gfCNCPoint3[13260] = {X 553.8289, Y 64.3705, Z -4.6667, A 0.000, B 0.000, C 0.000 }
gfCNCPoint3[13261] = {X 551.8531, Y 63.3648, Z -4.6667, A 0.000, B 0.000, C 0.000 }
gfCNCPoint3[13262] = {X 549.9931, Y 62.1583, Z -4.6667, A 0.000, B 0.000, C 0.000 }
gfCNCPoint3[13263] = {X 548.2693, Y 60.7642, Z -4.6667, A 0.000, B 0.000, C 0.000 }
gfCNCPoint3[13264] = {X 546.7005, Y 59.1977, Z -4.6667, A 0.000, B 0.000, C 0.000 }
gfCNCPoint3[13265] = {X 545.1840, Y 59.4175, Z -4.6667, A 0.000, B 0.000, C 0.000 }
gfCNCPoint3[13266] = {X 543.6528, Y 59.4759, Z -4.6667, A 0.000, B 0.000, C 0.000 }
gfCNCPoint3[13267] = {X 527.5783, Y 59.4763, Z -4.6667, A 0.000, B 0.000, C 0.000 }
gfCNCPoint3[13268] = {X 525.9215, Y 60.2766, Z -4.6667, A 0.000, B 0.000, C 0.000 }
gfCNCPoint3[13269] = {X 524.1774, Y 60.8627, Z -4.6667, A 0.000, B 0.000, C 0.000 }
gfCNCPoint3[13270] = {X 522.3736, Y 61.2254, Z -4.6667, A 0.000, B 0.000, C 0.000 }
gfCNCPoint3[13271] = {X 520.5385, Y 61.3590, Z -4.6667, A 0.000, B 0.000, C 0.000 }
gfCNCPoint3[13272] = {X 519.7998, Y 61.3591, Z -4.6667, A 0.000, B 0.000, C 0.000 }
gfCNCPoint3[13273] = {X 518.0043, Y 61.2474, Z -4.6667, A 0.000, B 0.000, C 0.000 }
gfCNCPoint3[13274] = {X 516.2365, Y 60.9138, Z -4.6667, A 0.000, B 0.000, C 0.000 }
gfCNCPoint3[13275] = {X 514.5237, Y 60.3637, Z -4.6667, A 0.000, B 0.000, C 0.000 }
gfCNCPoint3[13276] = {X 512.8923, Y 59.6054, Z -4.6667, A 0.000, B 0.000, C 0.000 }
gfCNCPoint3[13277] = {X 511.3676, Y 58.6507, Z -4.6667, A 0.000, B 0.000, C 0.000 }
gfCNCPoint3[13278] = {X 509.9730, Y 57.5142, Z -4.6667, A 0.000, B 0.000, C 0.000 }
gfCNCPoint3[13279] = {X 508.6156, Y 58.2113, Z -4.6667, A 0.000, B 0.000, C 0.000 }
gfCNCPoint3[13280] = {X 507.1924, Y 58.7617, Z -4.6667, A 0.000, B 0.000, C 0.000 }
gfCNCPoint3[13281] = {X 505.7192, Y 59.1593, Z -4.6667, A 0.000, B 0.000, C 0.000 }
gfCNCPoint3[13282] = {X 504.2123, Y 59.3996, Z -4.6667, A 0.000, B 0.000, C 0.000 }
gfCNCPoint3[13283] = {X 502.6885, Y 59.4800, Z -4.6667, A 0.000, B 0.000, C 0.000 }
gfCNCPoint3[13284] = {X 496.2450, Y 59.4800, Z -4.6667, A 0.000, B 0.000, C 0.000 }
gfCNCPoint3[13285] = {X 495.2580, Y 59.4463, Z -4.6667, A 0.000, B 0.000, C 0.000 }
gfCNCPoint3[13286] = {X 494.2756, Y 59.3454, Z -4.6667, A 0.000, B 0.000, C 0.000 }
gfCNCPoint3[13287] = {X 494.1342, Y 61.3005, Z -4.6667, A 0.000, B 0.000, C 0.000 }
gfCNCPoint3[13288] = {X 493.7950, Y 63.2312, Z -4.6667, A 0.000, B 0.000, C 0.000 }
gfCNCPoint3[13289] = {X 493.2616, Y 65.1174, Z -4.6667, A 0.000, B 0.000, C 0.000 }
gfCNCPoint3[13290] = {X 492.5393, Y 66.9397, Z -4.6667, A 0.000, B 0.000, C 0.000 }
gfCNCPoint3[13291] = {X 491.6358, Y 68.6792, Z -4.6667, A 0.000, B 0.000, C 0.000 }
gfCNCPoint3[13292] = {X 490.5603, Y 70.3180, Z -4.6667, A 0.000, B 0.000, C 0.000 }
gfCNCPoint3[13293] = {X 490.5605, Y 83.2950, Z -4.6667, A 0.000, B 0.000, C 0.000 }
gfCNCPoint3[13294] = {X 507.6815, Y 83.2950, Z -4.6667, A 0.000, B 0.000, C 0.000 }
gfCNCPoint3[13295] = {X 507.6815, Y 85.6950, Z -4.6667, A 0.000, B 0.000, C 0.000 }
gfCNCPoint3[13296] = {X 585.6966, Y 85.6950, Z -4.6667, A 0.000, B 0.000, C 0.000 }
gfCNCPoint3[13297] = {X 585.6966, Y 63.3150, Z -4.6667, A 0.000, B 0.000, C 0.000 }
gfCNCPoint3[13298] = {X 584.3995, Y 63.5678, Z -4.6667, A 0.000, B 0.000, C 0.000 }
gfCNCPoint3[13299] = {X 583.0880, Y 63.7288, Z -4.6667, A 0.000, B 0.000, C 0.000 }
gfCNCPoint3[13300] = {X 581.1243, Y 63.7971, Z -4.6667, A 0.000, B 0.000, C 0.000 }
gfCNCPoint3[13301] = {X 579.1642, Y 63.6600, Z -4.6667, A 0.000, B 0.000, C 0.000 }
gfCNCPoint3[13302] = {X 577.2291, Y 63.3191, Z -4.6667, A 0.000, B 0.000, C 0.000 }
gfCNCPoint3[13303] = {X 575.3401, Y 62.7781, Z -4.6667, A 0.000, B 0.000, C 0.000 }
gfCNCPoint3[13304] = {X 573.3441, Y 63.3435, Z -4.6667, A 0.000, B 0.000, C 0.000 }
gfCNCPoint3[13305] = {X 571.2979, Y 63.6855, Z -4.6667, A 0.000, B 0.000, C 0.000 }
gfCNCPoint3[13306] = {X 569.2264, Y 63.8000, Z -4.6667, A 0.000, B 0.000, C 0.000 }
gfCNCPoint3[13307] = {X 562.4443, Y 63.8000, Z -4.6667, A 0.000, B 0.000, C 0.000 }
gfCNCPoint3[13308] = {X 560.5408, Y 63.7034, Z -4.6667, A 0.000, B 0.000, C 0.000 }
gfCNCPoint3[13309] = {X 558.6568, Y 63.4145, Z -4.6667, A 0.000, B 0.000, C 0.000 }
gfCNCPoint3[13310] = {X 556.8118, Y 62.9364, Z -4.6667, A 0.000, B 0.000, C 0.000 }
gfCNCPoint3[13311] = {X 555.0247, Y 62.2739, Z -4.6667, A 0.000, B 0.000, C 0.000 }
gfCNCPoint3[13312] = {X 553.3138, Y 61.4339, Z -4.6667, A 0.000, B 0.000, C 0.000 }
gfCNCPoint3[13313] = {X 551.6968, Y 60.4250, Z -4.6667, A 0.000, B 0.000, C 0.000 }
gfCNCPoint3[13314] = {X 550.1902, Y 59.2575, Z -4.6667, A 0.000, B 0.000, C 0.000 }
gfCNCPoint3[13315] = {X 548.8096, Y 57.9435, Z -4.6667, A 0.000, B 0.000, C 0.000 }
gfCNCPoint3[13316] = {X 547.5691, Y 56.4965, Z -4.6667, A 0.000, B 0.000, C 0.000 }
gfCNCPoint3[13317] = {X 546.2936, Y 56.8314, Z -4.6667, A 0.000, B 0.000, C 0.000 }
gfCNCPoint3[13318] = {X 544.9891, Y 57.0253, Z -4.6667, A 0.000, B 0.000, C 0.000 }
gfCNCPoint3[13319] = {X 543.6713, Y 57.0759, Z -4.6667, A 0.000, B 0.000, C 0.000 }
gfCNCPoint3[13320] = {X 526.9187, Y 57.0763, Z -4.6667, A 0.000, B 0.000, C 0.000 }
gfCNCPoint3[13321] = {X 525.4335, Y 57.8746, Z -4.6667, A 0.000, B 0.000, C 0.000 }
gfCNCPoint3[13322] = {X 523.8527, Y 58.4612, Z -4.6667, A 0.000, B 0.000, C 0.000 }
gfCNCPoint3[13323] = {X 522.2063, Y 58.8250, Z -4.6667, A 0.000, B 0.000, C 0.000 }
gfCNCPoint3[13324] = {X 520.5255, Y 58.9590, Z -4.6667, A 0.000, B 0.000, C 0.000 }
gfCNCPoint3[13325] = {X 519.7998, Y 58.9591, Z -4.6667, A 0.000, B 0.000, C 0.000 }
gfCNCPoint3[13326] = {X 518.2467, Y 58.8589, Z -4.6667, A 0.000, B 0.000, C 0.000 }
gfCNCPoint3[13327] = {X 516.7195, Y 58.5598, Z -4.6667, A 0.000, B 0.000, C 0.000 }
gfCNCPoint3[13328] = {X 515.2433, Y 58.0668, Z -4.6667, A 0.000, B 0.000, C 0.000 }
gfCNCPoint3[13329] = {X 513.8428, Y 57.3882, Z -4.6667, A 0.000, B 0.000, C 0.000 }
gfCNCPoint3[13330] = {X 512.5411, Y 56.5351, Z -4.6667, A 0.000, B 0.000, C 0.000 }
gfCNCPoint3[13331] = {X 511.3600, Y 55.5218, Z -4.6667, A 0.000, B 0.000, C 0.000 }
gfCNCPoint3[13332] = {X 510.3189, Y 54.3650, Z -4.6667, A 0.000, B 0.000, C 0.000 }
gfCNCPoint3[13333] = {X 508.9711, Y 55.3177, Z -4.6667, A 0.000, B 0.000, C 0.000 }
gfCNCPoint3[13334] = {X 507.5060, Y 56.0778, Z -4.6667, A 0.000, B 0.000, C 0.000 }
gfCNCPoint3[13335] = {X 505.9510, Y 56.6311, Z -4.6667, A 0.000, B 0.000, C 0.000 }
gfCNCPoint3[13336] = {X 504.3351, Y 56.9672, Z -4.6667, A 0.000, B 0.000, C 0.000 }
gfCNCPoint3[13337] = {X 502.6885, Y 57.0800, Z -4.6667, A 0.000, B 0.000, C 0.000 }
gfCNCPoint3[13338] = {X 496.2450, Y 57.0800, Z -4.6667, A 0.000, B 0.000, C 0.000 }
gfCNCPoint3[13339] = {X 495.4216, Y 57.0519, Z -4.6667, A 0.000, B 0.000, C 0.000 }
gfCNCPoint3[13340] = {X 494.6020, Y 56.9677, Z -4.6667, A 0.000, B 0.000, C 0.000 }
gfCNCPoint3[13341] = {X 493.1719, Y 56.6826, Z -4.6667, A 0.000, B 0.000, C 0.000 }
gfCNCPoint3[13342] = {X 491.7866, Y 56.2272, Z -4.6667, A 0.000, B 0.000, C 0.000 }
gfCNCPoint3[13343] = {X 491.8566, Y 57.1124, Z -4.6667, A 0.000, B 0.000, C 0.000 }
gfCNCPoint3[13344] = {X 491.8800, Y 58.0000, Z -4.6667, A 0.000, B 0.000, C 0.000 }
gfCNCPoint3[13345] = {X 491.8794, Y 59.0735, Z -4.6667, A 0.000, B 0.000, C 0.000 }
gfCNCPoint3[13346] = {X 491.8781, Y 59.1839, Z -4.6667, A 0.000, B 0.000, C 0.000 }
gfCNCPoint3[13347] = {X 491.8762, Y 59.2942, Z -4.6667, A 0.000, B 0.000, C 0.000 }
gfCNCPoint3[13348] = {X 491.7363, Y 61.1318, Z -4.6667, A 0.000, B 0.000, C 0.000 }
gfCNCPoint3[13349] = {X 491.3970, Y 62.9431, Z -4.6667, A 0.000, B 0.000, C 0.000 }
gfCNCPoint3[13350] = {X 490.8623, Y 64.7067, Z -4.6667, A 0.000, B 0.000, C 0.000 }
gfCNCPoint3[13351] = {X 490.1385, Y 66.4014, Z -4.6667, A 0.000, B 0.000, C 0.000 }
gfCNCPoint3[13352] = {X 489.2342, Y 68.0072, Z -4.6667, A 0.000, B 0.000, C 0.000 }
gfCNCPoint3[13353] = {X 488.1603, Y 69.5048, Z -4.6667, A 0.000, B 0.000, C 0.000 }
gfCNCPoint3[13354] = {X 488.1606, Y 85.6950, Z -4.6667, A 0.000, B 0.000, C 0.000 }
gfCNCPoint3[13355] = {X 507.6815, Y 85.6950, Z -4.6667, A 0.000, B 0.000, C 0.000 }
gfCNCPoint3[13356] = {X 507.6815, Y 88.0950, Z -4.6667, A 0.000, B 0.000, C 0.000 }
gfCNCPoint3[13357] = {X 588.0966, Y 88.0950, Z -4.6667, A 0.000, B 0.000, C 0.000 }
gfCNCPoint3[13358] = {X 588.0966, Y 60.4644, Z -4.6667, A 0.000, B 0.000, C 0.000 }
gfCNCPoint3[13359] = {X 587.7998, Y 60.3564, Z -4.6667, A 0.000, B 0.000, C 0.000 }
gfCNCPoint3[13360] = {X 587.5052, Y 60.2427, Z -4.6667, A 0.000, B 0.000, C 0.000 }
gfCNCPoint3[13361] = {X 586.3439, Y 60.6540, Z -4.6667, A 0.000, B 0.000, C 0.000 }
gfCNCPoint3[13362] = {X 585.1550, Y 60.9769, Z -4.6667, A 0.000, B 0.000, C 0.000 }
gfCNCPoint3[13363] = {X 583.5153, Y 61.2699, Z -4.6667, A 0.000, B 0.000, C 0.000 }
gfCNCPoint3[13364] = {X 581.8543, Y 61.3951, Z -4.6667, A 0.000, B 0.000, C 0.000 }
gfCNCPoint3[13365] = {X 580.1893, Y 61.3512, Z -4.6667, A 0.000, B 0.000, C 0.000 }
gfCNCPoint3[13366] = {X 578.5372, Y 61.1386, Z -4.6667, A 0.000, B 0.000, C 0.000 }
gfCNCPoint3[13367] = {X 576.9153, Y 60.7595, Z -4.6667, A 0.000, B 0.000, C 0.000 }
gfCNCPoint3[13368] = {X 575.3401, Y 60.2178, Z -4.6667, A 0.000, B 0.000, C 0.000 }
gfCNCPoint3[13369] = {X 573.8611, Y 60.7315, Z -4.6667, A 0.000, B 0.000, C 0.000 }
gfCNCPoint3[13370] = {X 572.3399, Y 61.1017, Z -4.6667, A 0.000, B 0.000, C 0.000 }
gfCNCPoint3[13371] = {X 570.7903, Y 61.3253, Z -4.6667, A 0.000, B 0.000, C 0.000 }
gfCNCPoint3[13372] = {X 569.2264, Y 61.4000, Z -4.6667, A 0.000, B 0.000, C 0.000 }
gfCNCPoint3[13373] = {X 562.4443, Y 61.4000, Z -4.6667, A 0.000, B 0.000, C 0.000 }
gfCNCPoint3[13374] = {X 560.5829, Y 61.2940, Z -4.6667, A 0.000, B 0.000, C 0.000 }
gfCNCPoint3[13375] = {X 558.7455, Y 60.9774, Z -4.6667, A 0.000, B 0.000, C 0.000 }
gfCNCPoint3[13376] = {X 556.9559, Y 60.4544, Z -4.6667, A 0.000, B 0.000, C 0.000 }
gfCNCPoint3[13377] = {X 555.2372, Y 59.7315, Z -4.6667, A 0.000, B 0.000, C 0.000 }
gfCNCPoint3[13378] = {X 553.6118, Y 58.8183, Z -4.6667, A 0.000, B 0.000, C 0.000 }
gfCNCPoint3[13379] = {X 552.1004, Y 57.7265, Z -4.6667, A 0.000, B 0.000, C 0.000 }
gfCNCPoint3[13380] = {X 550.7228, Y 56.4702, Z -4.6667, A 0.000, B 0.000, C 0.000 }
gfCNCPoint3[13381] = {X 549.4966, Y 55.0657, Z -4.6667, A 0.000, B 0.000, C 0.000 }
gfCNCPoint3[13382] = {X 548.4378, Y 53.5310, Z -4.6667, A 0.000, B 0.000, C 0.000 }
gfCNCPoint3[13383] = {X 547.3159, Y 54.0426, Z -4.6667, A 0.000, B 0.000, C 0.000 }
gfCNCPoint3[13384] = {X 546.1381, Y 54.4074, Z -4.6667, A 0.000, B 0.000, C 0.000 }
gfCNCPoint3[13385] = {X 544.9235, Y 54.6197, Z -4.6667, A 0.000, B 0.000, C 0.000 }
gfCNCPoint3[13386] = {X 543.6918, Y 54.6759, Z -4.6667, A 0.000, B 0.000, C 0.000 }
gfCNCPoint3[13387] = {X 526.1843, Y 54.6763, Z -4.6667, A 0.000, B 0.000, C 0.000 }
gfCNCPoint3[13388] = {X 524.8902, Y 55.4730, Z -4.6667, A 0.000, B 0.000, C 0.000 }
gfCNCPoint3[13389] = {X 523.4888, Y 56.0608, Z -4.6667, A 0.000, B 0.000, C 0.000 }
gfCNCPoint3[13390] = {X 522.0136, Y 56.4257, Z -4.6667, A 0.000, B 0.000, C 0.000 }
gfCNCPoint3[13391] = {X 520.4998, Y 56.5591, Z -4.6667, A 0.000, B 0.000, C 0.000 }
gfCNCPoint3[13392] = {X 519.7998, Y 56.5591, Z -4.6667, A 0.000, B 0.000, C 0.000 }
gfCNCPoint3[13393] = {X 518.3493, Y 56.4498, Z -4.6667, A 0.000, B 0.000, C 0.000 }
gfCNCPoint3[13394] = {X 516.9316, Y 56.1244, Z -4.6667, A 0.000, B 0.000, C 0.000 }
gfCNCPoint3[13395] = {X 515.5787, Y 55.5903, Z -4.6667, A 0.000, B 0.000, C 0.000 }
gfCNCPoint3[13396] = {X 514.3210, Y 54.8595, Z -4.6667, A 0.000, B 0.000, C 0.000 }
gfCNCPoint3[13397] = {X 513.1871, Y 53.9484, Z -4.6667, A 0.000, B 0.000, C 0.000 }
gfCNCPoint3[13398] = {X 512.2025, Y 52.8778, Z -4.6667, A 0.000, B 0.000, C 0.000 }
gfCNCPoint3[13399] = {X 511.3855, Y 51.6648, Z -4.6667, A 0.000, B 0.000, C 0.000 }
gfCNCPoint3[13400] = {X 510.7606, Y 50.3426, Z -4.6667, A 0.000, B 0.000, C 0.000 }
gfCNCPoint3[13401] = {X 509.8636, Y 51.4977, Z -4.6667, A 0.000, B 0.000, C 0.000 }
gfCNCPoint3[13402] = {X 508.8029, Y 52.5044, Z -4.6667, A 0.000, B 0.000, C 0.000 }
gfCNCPoint3[13403] = {X 507.7229, Y 53.2678, Z -4.6667, A 0.000, B 0.000, C 0.000 }
gfCNCPoint3[13404] = {X 506.5489, Y 53.8769, Z -4.6667, A 0.000, B 0.000, C 0.000 }
gfCNCPoint3[13405] = {X 505.3028, Y 54.3203, Z -4.6667, A 0.000, B 0.000, C 0.000 }
gfCNCPoint3[13406] = {X 504.0080, Y 54.5896, Z -4.6667, A 0.000, B 0.000, C 0.000 }
gfCNCPoint3[13407] = {X 502.6885, Y 54.6800, Z -4.6667, A 0.000, B 0.000, C 0.000 }
gfCNCPoint3[13408] = {X 496.2450, Y 54.6800, Z -4.6667, A 0.000, B 0.000, C 0.000 }
gfCNCPoint3[13409] = {X 495.0285, Y 54.6033, Z -4.6667, A 0.000, B 0.000, C 0.000 }
gfCNCPoint3[13410] = {X 493.8313, Y 54.3742, Z -4.6667, A 0.000, B 0.000, C 0.000 }
gfCNCPoint3[13411] = {X 492.6724, Y 53.9966, Z -4.6667, A 0.000, B 0.000, C 0.000 }
gfCNCPoint3[13412] = {X 491.4451, Y 53.4062, Z -4.6667, A 0.000, B 0.000, C 0.000 }
gfCNCPoint3[13413] = {X 490.3129, Y 52.6493, Z -4.6667, A 0.000, B 0.000, C 0.000 }
gfCNCPoint3[13414] = {X 489.2980, Y 51.7410, Z -4.6667, A 0.000, B 0.000, C 0.000 }
gfCNCPoint3[13415] = {X 488.8683, Y 52.1573, Z -4.6667, A 0.000, B 0.000, C 0.000 }
gfCNCPoint3[13416] = {X 488.4137, Y 52.5463, Z -4.6667, A 0.000, B 0.000, C 0.000 }
gfCNCPoint3[13417] = {X 488.8649, Y 53.8245, Z -4.6667, A 0.000, B 0.000, C 0.000 }
gfCNCPoint3[13418] = {X 489.1946, Y 55.1393, Z -4.6667, A 0.000, B 0.000, C 0.000 }
gfCNCPoint3[13419] = {X 489.3999, Y 56.4792, Z -4.6667, A 0.000, B 0.000, C 0.000 }
gfCNCPoint3[13420] = {X 489.4600, Y 57.2386, Z -4.6667, A 0.000, B 0.000, C 0.000 }
gfCNCPoint3[13421] = {X 489.4800, Y 58.0000, Z -4.6667, A 0.000, B 0.000, C 0.000 }
gfCNCPoint3[13422] = {X 489.4795, Y 59.0537, Z -4.6667, A 0.000, B 0.000, C 0.000 }
gfCNCPoint3[13423] = {X 489.3596, Y 60.7977, Z -4.6667, A 0.000, B 0.000, C 0.000 }
gfCNCPoint3[13424] = {X 489.0303, Y 62.5146, Z -4.6667, A 0.000, B 0.000, C 0.000 }
gfCNCPoint3[13425] = {X 488.4966, Y 64.1793, Z -4.6667, A 0.000, B 0.000, C 0.000 }
gfCNCPoint3[13426] = {X 487.7661, Y 65.7676, Z -4.6667, A 0.000, B 0.000, C 0.000 }
gfCNCPoint3[13427] = {X 486.8496, Y 67.2562, Z -4.6667, A 0.000, B 0.000, C 0.000 }
gfCNCPoint3[13428] = {X 485.7603, Y 68.6236, Z -4.6667, A 0.000, B 0.000, C 0.000 }
gfCNCPoint3[13429] = {X 485.7606, Y 87.3794, Z -4.6667, A 0.000, B 0.000, C 0.000 }
gfCNCPoint3[13430] = {X 486.0686, Y 87.7323, Z -4.6667, A 0.000, B 0.000, C 0.000 }
gfCNCPoint3[13431] = {X 486.3650, Y 88.0950, Z -4.6667, A 0.000, B 0.000, C 0.000 }
gfCNCPoint3[13432] = {X 507.6815, Y 88.0950, Z -4.6667, A 0.000, B 0.000, C 0.000 }
gfCNCPoint3[13433] = {X 507.6815, Y 90.4950, Z -4.6667, A 0.000, B 0.000, C 0.000 }
gfCNCPoint3[13434] = {X 590.4966, Y 90.4950, Z -4.6667, A 0.000, B 0.000, C 0.000 }
gfCNCPoint3[13435] = {X 590.4966, Y 58.6615, Z -4.6667, A 0.000, B 0.000, C 0.000 }
gfCNCPoint3[13436] = {X 588.9715, Y 58.2279, Z -4.6667, A 0.000, B 0.000, C 0.000 }
gfCNCPoint3[13437] = {X 587.5052, Y 57.6246, Z -4.6667, A 0.000, B 0.000, C 0.000 }
gfCNCPoint3[13438] = {X 585.8387, Y 58.2956, Z -4.6667, A 0.000, B 0.000, C 0.000 }
gfCNCPoint3[13439] = {X 584.0999, Y 58.7477, Z -4.6667, A 0.000, B 0.000, C 0.000 }
gfCNCPoint3[13440] = {X 582.3176, Y 58.9733, Z -4.6667, A 0.000, B 0.000, C 0.000 }
gfCNCPoint3[13441] = {X 580.5210, Y 58.9689, Z -4.6667, A 0.000, B 0.000, C 0.000 }
gfCNCPoint3[13442] = {X 578.7398, Y 58.7344, Z -4.6667, A 0.000, B 0.000, C 0.000 }
gfCNCPoint3[13443] = {X 577.0034, Y 58.2738, Z -4.6667, A 0.000, B 0.000, C 0.000 }
gfCNCPoint3[13444] = {X 575.3401, Y 57.5945, Z -4.6667, A 0.000, B 0.000, C 0.000 }
gfCNCPoint3[13445] = {X 573.8813, Y 58.2035, Z -4.6667, A 0.000, B 0.000, C 0.000 }
gfCNCPoint3[13446] = {X 572.3630, Y 58.6441, Z -4.6667, A 0.000, B 0.000, C 0.000 }
gfCNCPoint3[13447] = {X 570.8048, Y 58.9107, Z -4.6667, A 0.000, B 0.000, C 0.000 }
gfCNCPoint3[13448] = {X 569.2264, Y 59.0000, Z -4.6667, A 0.000, B 0.000, C 0.000 }
gfCNCPoint3[13449] = {X 562.4443, Y 59.0000, Z -4.6667, A 0.000, B 0.000, C 0.000 }
gfCNCPoint3[13450] = {X 560.6577, Y 58.8855, Z -4.6667, A 0.000, B 0.000, C 0.000 }
gfCNCPoint3[13451] = {X 558.9002, Y 58.5440, Z -4.6667, A 0.000, B 0.000, C 0.000 }
gfCNCPoint3[13452] = {X 557.2008, Y 57.9810, Z -4.6667, A 0.000, B 0.000, C 0.000 }
gfCNCPoint3[13453] = {X 555.5870, Y 57.2057, Z -4.6667, A 0.000, B 0.000, C 0.000 }
gfCNCPoint3[13454] = {X 554.0855, Y 56.2307, Z -4.6667, A 0.000, B 0.000, C 0.000 }
gfCNCPoint3[13455] = {X 552.7206, Y 55.0722, Z -4.6667, A 0.000, B 0.000, C 0.000 }
gfCNCPoint3[13456] = {X 551.5147, Y 53.7489, Z -4.6667, A 0.000, B 0.000, C 0.000 }
gfCNCPoint3[13457] = {X 550.4875, Y 52.2826, Z -4.6667, A 0.000, B 0.000, C 0.000 }
gfCNCPoint3[13458] = {X 549.8378, Y 51.0889, Z -4.6667, A 0.000, B 0.000, C 0.000 }
gfCNCPoint3[13459] = {X 549.3068, Y 49.8379, Z -4.6667, A 0.000, B 0.000, C 0.000 }
gfCNCPoint3[13460] = {X 548.3754, Y 50.7147, Z -4.6667, A 0.000, B 0.000, C 0.000 }
gfCNCPoint3[13461] = {X 547.3051, Y 51.4151, Z -4.6667, A 0.000, B 0.000, C 0.000 }
gfCNCPoint3[13462] = {X 546.1635, Y 51.9061, Z -4.6667, A 0.000, B 0.000, C 0.000 }
gfCNCPoint3[13463] = {X 544.9551, Y 52.1958, Z -4.6667, A 0.000, B 0.000, C 0.000 }
gfCNCPoint3[13464] = {X 543.7151, Y 52.2759, Z -4.6667, A 0.000, B 0.000, C 0.000 }
gfCNCPoint3[13465] = {X 525.3422, Y 52.2763, Z -4.6667, A 0.000, B 0.000, C 0.000 }
gfCNCPoint3[13466] = {X 524.2750, Y 53.0678, Z -4.6667, A 0.000, B 0.000, C 0.000 }
gfCNCPoint3[13467] = {X 523.0840, Y 53.6568, Z -4.6667, A 0.000, B 0.000, C 0.000 }
gfCNCPoint3[13468] = {X 521.8072, Y 54.0245, Z -4.6667, A 0.000, B 0.000, C 0.000 }
gfCNCPoint3[13469] = {X 520.4853, Y 54.1591, Z -4.6667, A 0.000, B 0.000, C 0.000 }
gfCNCPoint3[13470] = {X 519.7998, Y 54.1591, Z -4.6667, A 0.000, B 0.000, C 0.000 }
gfCNCPoint3[13471] = {X 518.5529, Y 54.0515, Z -4.6667, A 0.000, B 0.000, C 0.000 }
gfCNCPoint3[13472] = {X 517.3428, Y 53.7320, Z -4.6667, A 0.000, B 0.000, C 0.000 }
gfCNCPoint3[13473] = {X 516.2054, Y 53.2099, Z -4.6667, A 0.000, B 0.000, C 0.000 }
gfCNCPoint3[13474] = {X 515.1742, Y 52.5007, Z -4.6667, A 0.000, B 0.000, C 0.000 }
gfCNCPoint3[13475] = {X 514.2797, Y 51.6254, Z -4.6667, A 0.000, B 0.000, C 0.000 }
gfCNCPoint3[13476] = {X 513.5483, Y 50.6098, Z -4.6667, A 0.000, B 0.000, C 0.000 }
gfCNCPoint3[13477] = {X 513.0017, Y 49.4839, Z -4.6667, A 0.000, B 0.000, C 0.000 }
gfCNCPoint3[13478] = {X 512.7353, Y 48.6374, Z -4.6667, A 0.000, B 0.000, C 0.000 }
gfCNCPoint3[13479] = {X 512.5739, Y 47.7649, Z -4.6667, A 0.000, B 0.000, C 0.000 }
gfCNCPoint3[13480] = {X 512.5198, Y 46.8791, Z -4.6667, A 0.000, B 0.000, C 0.000 }
gfCNCPoint3[13481] = {X 512.5198, Y 39.9011, Z -4.6667, A 0.000, B 0.000, C 0.000 }
gfCNCPoint3[13482] = {X 512.5807, Y 38.9610, Z -4.6667, A 0.000, B 0.000, C 0.000 }
gfCNCPoint3[13483] = {X 512.7626, Y 38.0366, Z -4.6667, A 0.000, B 0.000, C 0.000 }
gfCNCPoint3[13484] = {X 513.0623, Y 37.1434, Z -4.6667, A 0.000, B 0.000, C 0.000 }
gfCNCPoint3[13485] = {X 513.5579, Y 36.1545, Z -4.6667, A 0.000, B 0.000, C 0.000 }
gfCNCPoint3[13486] = {X 514.1976, Y 35.2520, Z -4.6667, A 0.000, B 0.000, C 0.000 }
gfCNCPoint3[13487] = {X 514.9666, Y 34.4569, Z -4.6667, A 0.000, B 0.000, C 0.000 }
gfCNCPoint3[13488] = {X 515.8472, Y 33.7875, Z -4.6667, A 0.000, B 0.000, C 0.000 }
gfCNCPoint3[13489] = {X 513.2412, Y 29.7566, Z -4.6667, A 0.000, B 0.000, C 0.000 }
gfCNCPoint3[13490] = {X 513.5216, Y 29.5807, Z -4.6667, A 0.000, B 0.000, C 0.000 }
gfCNCPoint3[13491] = {X 513.8068, Y 29.4125, Z -4.6667, A 0.000, B 0.000, C 0.000 }
gfCNCPoint3[13492] = {X 513.8068, Y 27.6757, Z -4.6667, A 0.000, B 0.000, C 0.000 }
gfCNCPoint3[13493] = {X 513.5215, Y 27.5011, Z -4.6667, A 0.000, B 0.000, C 0.000 }
gfCNCPoint3[13494] = {X 513.2412, Y 27.3187, Z -4.6667, A 0.000, B 0.000, C 0.000 }
gfCNCPoint3[13495] = {X 513.2412, Y 29.7566, Z -4.6667, A 0.000, B 0.000, C 0.000 }
gfCNCPoint3[13496] = {X 514.5442, Y 31.7721, Z -4.6667, A 0.000, B 0.000, C 0.000 }
gfCNCPoint3[13497] = {X 515.3547, Y 31.3021, Z -4.6667, A 0.000, B 0.000, C 0.000 }
gfCNCPoint3[13498] = {X 516.2068, Y 30.9126, Z -4.6667, A 0.000, B 0.000, C 0.000 }
gfCNCPoint3[13499] = {X 516.2068, Y 26.2046, Z -4.6667, A 0.000, B 0.000, C 0.000 }
gfCNCPoint3[13500] = {X 515.3712, Y 25.8040, Z -4.6667, A 0.000, B 0.000, C 0.000 }
gfCNCPoint3[13501] = {X 514.5778, Y 25.3254, Z -4.6667, A 0.000, B 0.000, C 0.000 }
gfCNCPoint3[13502] = {X 513.5946, Y 24.5705, Z -4.6667, A 0.000, B 0.000, C 0.000 }
gfCNCPoint3[13503] = {X 512.7159, Y 23.6962, Z -4.6667, A 0.000, B 0.000, C 0.000 }
gfCNCPoint3[13504] = {X 511.9562, Y 22.7167, Z -4.6667, A 0.000, B 0.000, C 0.000 }
gfCNCPoint3[13505] = {X 511.3278, Y 21.6481, Z -4.6667, A 0.000, B 0.000, C 0.000 }
gfCNCPoint3[13506] = {X 510.8412, Y 20.5081, Z -4.6667, A 0.000, B 0.000, C 0.000 }
gfCNCPoint3[13507] = {X 510.8411, Y 36.2343, Z -4.6667, A 0.000, B 0.000, C 0.000 }
gfCNCPoint3[13508] = {X 511.5001, Y 34.9193, Z -4.6667, A 0.000, B 0.000, C 0.000 }
gfCNCPoint3[13509] = {X 512.3507, Y 33.7194, Z -4.6667, A 0.000, B 0.000, C 0.000 }
gfCNCPoint3[13510] = {X 513.3733, Y 32.6622, Z -4.6667, A 0.000, B 0.000, C 0.000 }
gfCNCPoint3[13511] = {X 514.5442, Y 31.7721, Z -4.6667, A 0.000, B 0.000, C 0.000 }
gfCNCPoint3[13512] = {X 515.8472, Y 33.7875, Z -4.6667, A 0.000, B 0.000, C 0.000 }
gfCNCPoint3[13513] = {X 516.7437, Y 33.2936, Z -4.6667, A 0.000, B 0.000, C 0.000 }
gfCNCPoint3[13514] = {X 517.7006, Y 32.9303, Z -4.6667, A 0.000, B 0.000, C 0.000 }
gfCNCPoint3[13515] = {X 518.6990, Y 32.7048, Z -4.6667, A 0.000, B 0.000, C 0.000 }
gfCNCPoint3[13516] = {X 518.6299, Y 32.1290, Z -4.6667, A 0.000, B 0.000, C 0.000 }
gfCNCPoint3[13517] = {X 518.6068, Y 31.5494, Z -4.6667, A 0.000, B 0.000, C 0.000 }
gfCNCPoint3[13518] = {X 518.6068, Y 24.5714, Z -4.6667, A 0.000, B 0.000, C 0.000 }
gfCNCPoint3[13519] = {X 518.6080, Y 24.4373, Z -4.6667, A 0.000, B 0.000, C 0.000 }
gfCNCPoint3[13520] = {X 517.3912, Y 24.0940, Z -4.6667, A 0.000, B 0.000, C 0.000 }
gfCNCPoint3[13521] = {X 516.2521, Y 23.5453, Z -4.6667, A 0.000, B 0.000, C 0.000 }
gfCNCPoint3[13522] = {X 515.2251, Y 22.8078, Z -4.6667, A 0.000, B 0.000, C 0.000 }
gfCNCPoint3[13523] = {X 514.3412, Y 21.9037, Z -4.6667, A 0.000, B 0.000, C 0.000 }
gfCNCPoint3[13524] = {X 513.6271, Y 20.8603, Z -4.6667, A 0.000, B 0.000, C 0.000 }
gfCNCPoint3[13525] = {X 513.1043, Y 19.7091, Z -4.6667, A 0.000, B 0.000, C 0.000 }
gfCNCPoint3[13526] = {X 512.7937, Y 18.5151, Z -4.6667, A 0.000, B 0.000, C 0.000 }
gfCNCPoint3[13527] = {X 512.6891, Y 17.2857, Z -4.6667, A 0.000, B 0.000, C 0.000 }
gfCNCPoint3[13528] = {X 512.6891, Y 10.3077, Z -4.6667, A 0.000, B 0.000, C 0.000 }
gfCNCPoint3[13529] = {X 512.7002, Y 9.9057, Z -4.6667, A 0.000, B 0.000, C 0.000 }
gfCNCPoint3[13530] = {X 512.7335, Y 9.5050, Z -4.6667, A 0.000, B 0.000, C 0.000 }
gfCNCPoint3[13531] = {X 509.4590, Y 9.5050, Z -4.6667, A 0.000, B 0.000, C 0.000 }
gfCNCPoint3[13532] = {X 509.7405, Y 10.3720, Z -4.6667, A 0.000, B 0.000, C 0.000 }
gfCNCPoint3[13533] = {X 509.9113, Y 11.2675, Z -4.6667, A 0.000, B 0.000, C 0.000 }
gfCNCPoint3[13534] = {X 509.9685, Y 12.1773, Z -4.6667, A 0.000, B 0.000, C 0.000 }
gfCNCPoint3[13535] = {X 509.9682, Y 13.0462, Z -4.6667, A 0.000, B 0.000, C 0.000 }
gfCNCPoint3[13536] = {X 509.8611, Y 14.2235, Z -4.6667, A 0.000, B 0.000, C 0.000 }
gfCNCPoint3[13537] = {X 509.5650, Y 15.3681, Z -4.6667, A 0.000, B 0.000, C 0.000 }
gfCNCPoint3[13538] = {X 509.0875, Y 16.4496, Z -4.6667, A 0.000, B 0.000, C 0.000 }
gfCNCPoint3[13539] = {X 508.4412, Y 17.4395, Z -4.6667, A 0.000, B 0.000, C 0.000 }
gfCNCPoint3[13540] = {X 508.4411, Y 39.7472, Z -4.6667, A 0.000, B 0.000, C 0.000 }
gfCNCPoint3[13541] = {X 509.0892, Y 40.7405, Z -4.6667, A 0.000, B 0.000, C 0.000 }
gfCNCPoint3[13542] = {X 509.5674, Y 41.8259, Z -4.6667, A 0.000, B 0.000, C 0.000 }
gfCNCPoint3[13543] = {X 509.8631, Y 42.9744, Z -4.6667, A 0.000, B 0.000, C 0.000 }
gfCNCPoint3[13544] = {X 509.9683, Y 44.1558, Z -4.6667, A 0.000, B 0.000, C 0.000 }
gfCNCPoint3[13545] = {X 509.9685, Y 45.0000, Z -4.6667, A 0.000, B 0.000, C 0.000 }
gfCNCPoint3[13546] = {X 509.8909, Y 46.0603, Z -4.6667, A 0.000, B 0.000, C 0.000 }
gfCNCPoint3[13547] = {X 509.6596, Y 47.0980, Z -4.6667, A 0.000, B 0.000, C 0.000 }
gfCNCPoint3[13548] = {X 509.2797, Y 48.0910, Z -4.6667, A 0.000, B 0.000, C 0.000 }
gfCNCPoint3[13549] = {X 508.7593, Y 49.0180, Z -4.6667, A 0.000, B 0.000, C 0.000 }
gfCNCPoint3[13550] = {X 508.0200, Y 49.9571, Z -4.6667, A 0.000, B 0.000, C 0.000 }
gfCNCPoint3[13551] = {X 507.1371, Y 50.7626, Z -4.6667, A 0.000, B 0.000, C 0.000 }
gfCNCPoint3[13552] = {X 506.1343, Y 51.4129, Z -4.6667, A 0.000, B 0.000, C 0.000 }
gfCNCPoint3[13553] = {X 505.0386, Y 51.8902, Z -4.6667, A 0.000, B 0.000, C 0.000 }
gfCNCPoint3[13554] = {X 503.8796, Y 52.1819, Z -4.6667, A 0.000, B 0.000, C 0.000 }
gfCNCPoint3[13555] = {X 502.6885, Y 52.2800, Z -4.6667, A 0.000, B 0.000, C 0.000 }
gfCNCPoint3[13556] = {X 496.2450, Y 52.2800, Z -4.6667, A 0.000, B 0.000, C 0.000 }
gfCNCPoint3[13557] = {X 495.0845, Y 52.1869, Z -4.6667, A 0.000, B 0.000, C 0.000 }
gfCNCPoint3[13558] = {X 493.9538, Y 51.9100, Z -4.6667, A 0.000, B 0.000, C 0.000 }
gfCNCPoint3[13559] = {X 492.8816, Y 51.4564, Z -4.6667, A 0.000, B 0.000, C 0.000 }
gfCNCPoint3[13560] = {X 491.8954, Y 50.8377, Z -4.6667, A 0.000, B 0.000, C 0.000 }
gfCNCPoint3[13561] = {X 491.0204, Y 50.0697, Z -4.6667, A 0.000, B 0.000, C 0.000 }
gfCNCPoint3[13562] = {X 490.2980, Y 49.1989, Z -4.6667, A 0.000, B 0.000, C 0.000 }
gfCNCPoint3[13563] = {X 489.7192, Y 48.2267, Z -4.6667, A 0.000, B 0.000, C 0.000 }
gfCNCPoint3[13564] = {X 489.2980, Y 47.1766, Z -4.6667, A 0.000, B 0.000, C 0.000 }
gfCNCPoint3[13565] = {X 488.8769, Y 48.2267, Z -4.6667, A 0.000, B 0.000, C 0.000 }
gfCNCPoint3[13566] = {X 488.2981, Y 49.1989, Z -4.6667, A 0.000, B 0.000, C 0.000 }
gfCNCPoint3[13567] = {X 487.5756, Y 50.0697, Z -4.6667, A 0.000, B 0.000, C 0.000 }
gfCNCPoint3[13568] = {X 486.8824, Y 50.6978, Z -4.6667, A 0.000, B 0.000, C 0.000 }
gfCNCPoint3[13569] = {X 486.1145, Y 51.2318, Z -4.6667, A 0.000, B 0.000, C 0.000 }
gfCNCPoint3[13570] = {X 485.2843, Y 51.6629, Z -4.6667, A 0.000, B 0.000, C 0.000 }
gfCNCPoint3[13571] = {X 486.0586, Y 53.1385, Z -4.6667, A 0.000, B 0.000, C 0.000 }
gfCNCPoint3[13572] = {X 486.6224, Y 54.7067, Z -4.6667, A 0.000, B 0.000, C 0.000 }
gfCNCPoint3[13573] = {X 486.9651, Y 56.3375, Z -4.6667, A 0.000, B 0.000, C 0.000 }
gfCNCPoint3[13574] = {X 487.0800, Y 58.0000, Z -4.6667, A 0.000, B 0.000, C 0.000 }
gfCNCPoint3[13575] = {X 487.0796, Y 59.0339, Z -4.6667, A 0.000, B 0.000, C 0.000 }
gfCNCPoint3[13576] = {X 486.9596, Y 60.6352, Z -4.6667, A 0.000, B 0.000, C 0.000 }
gfCNCPoint3[13577] = {X 486.6283, Y 62.2064, Z -4.6667, A 0.000, B 0.000, C 0.000 }
gfCNCPoint3[13578] = {X 486.0916, Y 63.7199, Z -4.6667, A 0.000, B 0.000, C 0.000 }
gfCNCPoint3[13579] = {X 485.3588, Y 65.1487, Z -4.6667, A 0.000, B 0.000, C 0.000 }
gfCNCPoint3[13580] = {X 484.4430, Y 66.4678, Z -4.6667, A 0.000, B 0.000, C 0.000 }
gfCNCPoint3[13581] = {X 483.3603, Y 67.6537, Z -4.6667, A 0.000, B 0.000, C 0.000 }
gfCNCPoint3[13582] = {X 483.3606, Y 88.3504, Z -4.6667, A 0.000, B 0.000, C 0.000 }
gfCNCPoint3[13583] = {X 484.3106, Y 89.3713, Z -4.6667, A 0.000, B 0.000, C 0.000 }
gfCNCPoint3[13584] = {X 485.1364, Y 90.4950, Z -4.6667, A 0.000, B 0.000, C 0.000 }
gfCNCPoint3[13585] = {X 507.6815, Y 90.4950, Z -4.6667, A 0.000, B 0.000, C 0.000 }
gfCNCPoint3[13586] = {X 507.6815, Y 92.8950, Z -4.6667, A 0.000, B 0.000, C 0.000 }
gfCNCPoint3[13587] = {X 592.8966, Y 92.8950, Z -4.6667, A 0.000, B 0.000, C 0.000 }
gfCNCPoint3[13588] = {X 592.8966, Y 56.5812, Z -4.6667, A 0.000, B 0.000, C 0.000 }
gfCNCPoint3[13589] = {X 591.4810, Y 56.4128, Z -4.6667, A 0.000, B 0.000, C 0.000 }
gfCNCPoint3[13590] = {X 590.0968, Y 56.0720, Z -4.6667, A 0.000, B 0.000, C 0.000 }
gfCNCPoint3[13591] = {X 588.7648, Y 55.5641, Z -4.6667, A 0.000, B 0.000, C 0.000 }
gfCNCPoint3[13592] = {X 587.5052, Y 54.8965, Z -4.6667, A 0.000, B 0.000, C 0.000 }
gfCNCPoint3[13593] = {X 586.9690, Y 55.2051, Z -4.6667, A 0.000, B 0.000, C 0.000 }
gfCNCPoint3[13594] = {X 586.4171, Y 55.4846, Z -4.6667, A 0.000, B 0.000, C 0.000 }
gfCNCPoint3[13595] = {X 584.8782, Y 56.0830, Z -4.6667, A 0.000, B 0.000, C 0.000 }
gfCNCPoint3[13596] = {X 583.2699, Y 56.4570, Z -4.6667, A 0.000, B 0.000, C 0.000 }
gfCNCPoint3[13597] = {X 581.6248, Y 56.5987, Z -4.6667, A 0.000, B 0.000, C 0.000 }
gfCNCPoint3[13598] = {X 579.9763, Y 56.5055, Z -4.6667, A 0.000, B 0.000, C 0.000 }
gfCNCPoint3[13599] = {X 578.3577, Y 56.1792, Z -4.6667, A 0.000, B 0.000, C 0.000 }
gfCNCPoint3[13600] = {X 576.8018, Y 55.6263, Z -4.6667, A 0.000, B 0.000, C 0.000 }
gfCNCPoint3[13601] = {X 575.3401, Y 54.8581, Z -4.6667, A 0.000, B 0.000, C 0.000 }
gfCNCPoint3[13602] = {X 573.9176, Y 55.6091, Z -4.6667, A 0.000, B 0.000, C 0.000 }
gfCNCPoint3[13603] = {X 572.4049, Y 56.1560, Z -4.6667, A 0.000, B 0.000, C 0.000 }
gfCNCPoint3[13604] = {X 570.8311, Y 56.4885, Z -4.6667, A 0.000, B 0.000, C 0.000 }
gfCNCPoint3[13605] = {X 569.2264, Y 56.6000, Z -4.6667, A 0.000, B 0.000, C 0.000 }
gfCNCPoint3[13606] = {X 562.4443, Y 56.6000, Z -4.6667, A 0.000, B 0.000, C 0.000 }
gfCNCPoint3[13607] = {X 560.8793, Y 56.4939, Z -4.6667, A 0.000, B 0.000, C 0.000 }
gfCNCPoint3[13608] = {X 559.3429, Y 56.1777, Z -4.6667, A 0.000, B 0.000, C 0.000 }
gfCNCPoint3[13609] = {X 557.8632, Y 55.6571, Z -4.6667, A 0.000, B 0.000, C 0.000 }
gfCNCPoint3[13610] = {X 556.4673, Y 54.9416, Z -4.6667, A 0.000, B 0.000, C 0.000 }
gfCNCPoint3[13611] = {X 555.1806, Y 54.0443, Z -4.6667, A 0.000, B 0.000, C 0.000 }
gfCNCPoint3[13612] = {X 554.0268, Y 52.9816, Z -4.6667, A 0.000, B 0.000, C 0.000 }
gfCNCPoint3[13613] = {X 553.0269, Y 51.7730, Z -4.6667, A 0.000, B 0.000, C 0.000 }
gfCNCPoint3[13614] = {X 552.1993, Y 50.4405, Z -4.6667, A 0.000, B 0.000, C 0.000 }
gfCNCPoint3[13615] = {X 551.5589, Y 49.0085, Z -4.6667, A 0.000, B 0.000, C 0.000 }
gfCNCPoint3[13616] = {X 551.1637, Y 47.7035, Z -4.6667, A 0.000, B 0.000, C 0.000 }
gfCNCPoint3[13617] = {X 550.9244, Y 46.3612, Z -4.6667, A 0.000, B 0.000, C 0.000 }
gfCNCPoint3[13618] = {X 550.8443, Y 45.0000, Z -4.6667, A 0.000, B 0.000, C 0.000 }
gfCNCPoint3[13619] = {X 550.8444, Y 44.0347, Z -4.6667, A 0.000, B 0.000, C 0.000 }
gfCNCPoint3[13620] = {X 550.9587, Y 42.4546, Z -4.6667, A 0.000, B 0.000, C 0.000 }
gfCNCPoint3[13621] = {X 551.2867, Y 40.9046, Z -4.6667, A 0.000, B 0.000, C 0.000 }
gfCNCPoint3[13622] = {X 551.8223, Y 39.4136, Z -4.6667, A 0.000, B 0.000, C 0.000 }
gfCNCPoint3[13623] = {X 549.6240, Y 38.4504, Z -4.6667, A 0.000, B 0.000, C 0.000 }
gfCNCPoint3[13624] = {X 549.7926, Y 38.0804, Z -4.6667, A 0.000, B 0.000, C 0.000 }
gfCNCPoint3[13625] = {X 549.9718, Y 37.7155, Z -4.6667, A 0.000, B 0.000, C 0.000 }
gfCNCPoint3[13626] = {X 549.9718, Y 16.9509, Z -4.6667, A 0.000, B 0.000, C 0.000 }
gfCNCPoint3[13627] = {X 549.8028, Y 17.1990, Z -4.6667, A 0.000, B 0.000, C 0.000 }
gfCNCPoint3[13628] = {X 549.6238, Y 17.4399, Z -4.6667, A 0.000, B 0.000, C 0.000 }
gfCNCPoint3[13629] = {X 549.6240, Y 38.4504, Z -4.6667, A 0.000, B 0.000, C 0.000 }
gfCNCPoint3[13630] = {X 551.8223, Y 39.4136, Z -4.6667, A 0.000, B 0.000, C 0.000 }
gfCNCPoint3[13631] = {X 552.0826, Y 38.8595, Z -4.6667, A 0.000, B 0.000, C 0.000 }
gfCNCPoint3[13632] = {X 552.3718, Y 38.3199, Z -4.6667, A 0.000, B 0.000, C 0.000 }
gfCNCPoint3[13633] = {X 552.3718, Y 11.6877, Z -4.6667, A 0.000, B 0.000, C 0.000 }
gfCNCPoint3[13634] = {X 551.6705, Y 10.2335, Z -4.6667, A 0.000, B 0.000, C 0.000 }
gfCNCPoint3[13635] = {X 551.1779, Y 8.6960, Z -4.6667, A 0.000, B 0.000, C 0.000 }
gfCNCPoint3[13636] = {X 550.9035, Y 7.1050, Z -4.6667, A 0.000, B 0.000, C 0.000 }
gfCNCPoint3[13637] = {X 524.2928, Y 7.1050, Z -4.6667, A 0.000, B 0.000, C 0.000 }
gfCNCPoint3[13638] = {X 524.3786, Y 7.2064, Z -4.6667, A 0.000, B 0.000, C 0.000 }
gfCNCPoint3[13639] = {X 524.4616, Y 7.3101, Z -4.6667, A 0.000, B 0.000, C 0.000 }
gfCNCPoint3[13640] = {X 543.7426, Y 7.3106, Z -4.6667, A 0.000, B 0.000, C 0.000 }
gfCNCPoint3[13641] = {X 544.7119, Y 7.3827, Z -4.6667, A 0.000, B 0.000, C 0.000 }
gfCNCPoint3[13642] = {X 545.6477, Y 7.6453, Z -4.6667, A 0.000, B 0.000, C 0.000 }
gfCNCPoint3[13643] = {X 546.5130, Y 8.0880, Z -4.6667, A 0.000, B 0.000, C 0.000 }
gfCNCPoint3[13644] = {X 547.2735, Y 8.6932, Z -4.6667, A 0.000, B 0.000, C 0.000 }
gfCNCPoint3[13645] = {X 547.8992, Y 9.4370, Z -4.6667, A 0.000, B 0.000, C 0.000 }
gfCNCPoint3[13646] = {X 548.3652, Y 10.2900, Z -4.6667, A 0.000, B 0.000, C 0.000 }
gfCNCPoint3[13647] = {X 548.6530, Y 11.2184, Z -4.6667, A 0.000, B 0.000, C 0.000 }
gfCNCPoint3[13648] = {X 548.7514, Y 12.1853, Z -4.6667, A 0.000, B 0.000, C 0.000 }
gfCNCPoint3[13649] = {X 548.7514, Y 12.9780, Z -4.6667, A 0.000, B 0.000, C 0.000 }
gfCNCPoint3[13650] = {X 548.6614, Y 13.9112, Z -4.6667, A 0.000, B 0.000, C 0.000 }
gfCNCPoint3[13651] = {X 548.3945, Y 14.8100, Z -4.6667, A 0.000, B 0.000, C 0.000 }
gfCNCPoint3[13652] = {X 547.9607, Y 15.6412, Z -4.6667, A 0.000, B 0.000, C 0.000 }
gfCNCPoint3[13653] = {X 547.6183, Y 16.1045, Z -4.6667, A 0.000, B 0.000, C 0.000 }
gfCNCPoint3[13654] = {X 547.2238, Y 16.5243, Z -4.6667, A 0.000, B 0.000, C 0.000 }
gfCNCPoint3[13655] = {X 547.2240, Y 40.6628, Z -4.6667, A 0.000, B 0.000, C 0.000 }
gfCNCPoint3[13656] = {X 547.8654, Y 41.4047, Z -4.6667, A 0.000, B 0.000, C 0.000 }
gfCNCPoint3[13657] = {X 548.3454, Y 42.2599, Z -4.6667, A 0.000, B 0.000, C 0.000 }
gfCNCPoint3[13658] = {X 548.6447, Y 43.1938, Z -4.6667, A 0.000, B 0.000, C 0.000 }
gfCNCPoint3[13659] = {X 548.7513, Y 44.1687, Z -4.6667, A 0.000, B 0.000, C 0.000 }
gfCNCPoint3[13660] = {X 548.7514, Y 45.0006, Z -4.6667, A 0.000, B 0.000, C 0.000 }
gfCNCPoint3[13661] = {X 548.6698, Y 45.8823, Z -4.6667, A 0.000, B 0.000, C 0.000 }
gfCNCPoint3[13662] = {X 548.4304, Y 46.7347, Z -4.6667, A 0.000, B 0.000, C 0.000 }
gfCNCPoint3[13663] = {X 548.0410, Y 47.5299, Z -4.6667, A 0.000, B 0.000, C 0.000 }
gfCNCPoint3[13664] = {X 547.5145, Y 48.2417, Z -4.6667, A 0.000, B 0.000, C 0.000 }
gfCNCPoint3[13665] = {X 546.7289, Y 48.9513, Z -4.6667, A 0.000, B 0.000, C 0.000 }
gfCNCPoint3[13666] = {X 545.8088, Y 49.4749, Z -4.6667, A 0.000, B 0.000, C 0.000 }
gfCNCPoint3[13667] = {X 544.7976, Y 49.7881, Z -4.6667, A 0.000, B 0.000, C 0.000 }
gfCNCPoint3[13668] = {X 543.7426, Y 49.8759, Z -4.6667, A 0.000, B 0.000, C 0.000 }
gfCNCPoint3[13669] = {X 524.3235, Y 49.8764, Z -4.6667, A 0.000, B 0.000, C 0.000 }
gfCNCPoint3[13670] = {X 523.7107, Y 50.5152, Z -4.6667, A 0.000, B 0.000, C 0.000 }
gfCNCPoint3[13671] = {X 522.9955, Y 51.0370, Z -4.6667, A 0.000, B 0.000, C 0.000 }
gfCNCPoint3[13672] = {X 522.2000, Y 51.4255, Z -4.6667, A 0.000, B 0.000, C 0.000 }
gfCNCPoint3[13673] = {X 521.3488, Y 51.6687, Z -4.6667, A 0.000, B 0.000, C 0.000 }
gfCNCPoint3[13674] = {X 520.4681, Y 51.7591, Z -4.6667, A 0.000, B 0.000, C 0.000 }
gfCNCPoint3[13675] = {X 519.7998, Y 51.7591, Z -4.6667, A 0.000, B 0.000, C 0.000 }
gfCNCPoint3[13676] = {X 518.8477, Y 51.6654, Z -4.6667, A 0.000, B 0.000, C 0.000 }
gfCNCPoint3[13677] = {X 517.9323, Y 51.3877, Z -4.6667, A 0.000, B 0.000, C 0.000 }
gfCNCPoint3[13678] = {X 517.0886, Y 50.9367, Z -4.6667, A 0.000, B 0.000, C 0.000 }
gfCNCPoint3[13679] = {X 516.3491, Y 50.3298, Z -4.6667, A 0.000, B 0.000, C 0.000 }
gfCNCPoint3[13680] = {X 515.7422, Y 49.5903, Z -4.6667, A 0.000, B 0.000, C 0.000 }
gfCNCPoint3[13681] = {X 515.2912, Y 48.7466, Z -4.6667, A 0.000, B 0.000, C 0.000 }
gfCNCPoint3[13682] = {X 515.0135, Y 47.8312, Z -4.6667, A 0.000, B 0.000, C 0.000 }
gfCNCPoint3[13683] = {X 514.9198, Y 46.8791, Z -4.6667, A 0.000, B 0.000, C 0.000 }
gfCNCPoint3[13684] = {X 514.9198, Y 39.9011, Z -4.6667, A 0.000, B 0.000, C 0.000 }
gfCNCPoint3[13685] = {X 515.0197, Y 38.9186, Z -4.6667, A 0.000, B 0.000, C 0.000 }
gfCNCPoint3[13686] = {X 515.3154, Y 37.9764, Z -4.6667, A 0.000, B 0.000, C 0.000 }
gfCNCPoint3[13687] = {X 515.7947, Y 37.1129, Z -4.6667, A 0.000, B 0.000, C 0.000 }
gfCNCPoint3[13688] = {X 516.4381, Y 36.3637, Z -4.6667, A 0.000, B 0.000, C 0.000 }
gfCNCPoint3[13689] = {X 517.2191, Y 35.7593, Z -4.6667, A 0.000, B 0.000, C 0.000 }
gfCNCPoint3[13690] = {X 518.1058, Y 35.3245, Z -4.6667, A 0.000, B 0.000, C 0.000 }
gfCNCPoint3[13691] = {X 519.0619, Y 35.0772, Z -4.6667, A 0.000, B 0.000, C 0.000 }
gfCNCPoint3[13692] = {X 519.4084, Y 35.0368, Z -4.6667, A 0.000, B 0.000, C 0.000 }
gfCNCPoint3[13693] = {X 519.7568, Y 35.0213, Z -4.6667, A 0.000, B 0.000, C 0.000 }
gfCNCPoint3[13694] = {X 520.5345, Y 35.0216, Z -4.6667, A 0.000, B 0.000, C 0.000 }
gfCNCPoint3[13695] = {X 521.4084, Y 35.1125, Z -4.6667, A 0.000, B 0.000, C 0.000 }
gfCNCPoint3[13696] = {X 522.2519, Y 35.3588, Z -4.6667, A 0.000, B 0.000, C 0.000 }
gfCNCPoint3[13697] = {X 523.0375, Y 35.7523, Z -4.6667, A 0.000, B 0.000, C 0.000 }
gfCNCPoint3[13698] = {X 523.7399, Y 36.2802, Z -4.6667, A 0.000, B 0.000, C 0.000 }
gfCNCPoint3[13699] = {X 524.3361, Y 36.9256, Z -4.6667, A 0.000, B 0.000, C 0.000 }
gfCNCPoint3[13700] = {X 534.0719, Y 36.9260, Z -4.6667, A 0.000, B 0.000, C 0.000 }
gfCNCPoint3[13701] = {X 534.0719, Y 34.5254, Z -4.6667, A 0.000, B 0.000, C 0.000 }
gfCNCPoint3[13702] = {X 530.3962, Y 34.5251, Z -4.6667, A 0.000, B 0.000, C 0.000 }
gfCNCPoint3[13703] = {X 529.7963, Y 35.1737, Z -4.6667, A 0.000, B 0.000, C 0.000 }
gfCNCPoint3[13704] = {X 529.0893, Y 35.7035, Z -4.6667, A 0.000, B 0.000, C 0.000 }
gfCNCPoint3[13705] = {X 528.2984, Y 36.0972, Z -4.6667, A 0.000, B 0.000, C 0.000 }
gfCNCPoint3[13706] = {X 527.4494, Y 36.3418, Z -4.6667, A 0.000, B 0.000, C 0.000 }
gfCNCPoint3[13707] = {X 526.5703, Y 36.4293, Z -4.6667, A 0.000, B 0.000, C 0.000 }
gfCNCPoint3[13708] = {X 525.8868, Y 36.4294, Z -4.6667, A 0.000, B 0.000, C 0.000 }
gfCNCPoint3[13709] = {X 524.9094, Y 36.3306, Z -4.6667, A 0.000, B 0.000, C 0.000 }
gfCNCPoint3[13710] = {X 523.9717, Y 36.0380, Z -4.6667, A 0.000, B 0.000, C 0.000 }
gfCNCPoint3[13711] = {X 523.1116, Y 35.5636, Z -4.6667, A 0.000, B 0.000, C 0.000 }
gfCNCPoint3[13712] = {X 522.3639, Y 34.9265, Z -4.6667, A 0.000, B 0.000, C 0.000 }
gfCNCPoint3[13713] = {X 521.7590, Y 34.1525, Z -4.6667, A 0.000, B 0.000, C 0.000 }
gfCNCPoint3[13714] = {X 521.3213, Y 33.2731, Z -4.6667, A 0.000, B 0.000, C 0.000 }
gfCNCPoint3[13715] = {X 521.0686, Y 32.3239, Z -4.6667, A 0.000, B 0.000, C 0.000 }
gfCNCPoint3[13716] = {X 521.0222, Y 31.9379, Z -4.6667, A 0.000, B 0.000, C 0.000 }
gfCNCPoint3[13717] = {X 521.0068, Y 31.5494, Z -4.6667, A 0.000, B 0.000, C 0.000 }
gfCNCPoint3[13718] = {X 521.0076, Y 24.4815, Z -4.6667, A 0.000, B 0.000, C 0.000 }
gfCNCPoint3[13719] = {X 521.0984, Y 23.6300, Z -4.6667, A 0.000, B 0.000, C 0.000 }
gfCNCPoint3[13720] = {X 521.3368, Y 22.8074, Z -4.6667, A 0.000, B 0.000, C 0.000 }
gfCNCPoint3[13721] = {X 521.7152, Y 22.0391, Z -4.6667, A 0.000, B 0.000, C 0.000 }
gfCNCPoint3[13722] = {X 521.1864, Y 22.1316, Z -4.6667, A 0.000, B 0.000, C 0.000 }
gfCNCPoint3[13723] = {X 520.6505, Y 22.1656, Z -4.6667, A 0.000, B 0.000, C 0.000 }
gfCNCPoint3[13724] = {X 519.9691, Y 22.1657, Z -4.6667, A 0.000, B 0.000, C 0.000 }
gfCNCPoint3[13725] = {X 519.5109, Y 22.1442, Z -4.6667, A 0.000, B 0.000, C 0.000 }
gfCNCPoint3[13726] = {X 519.0567, Y 22.0797, Z -4.6667, A 0.000, B 0.000, C 0.000 }
gfCNCPoint3[13727] = {X 518.1336, Y 21.8074, Z -4.6667, A 0.000, B 0.000, C 0.000 }
gfCNCPoint3[13728] = {X 517.2820, Y 21.3592, Z -4.6667, A 0.000, B 0.000, C 0.000 }
gfCNCPoint3[13729] = {X 516.5348, Y 20.7527, Z -4.6667, A 0.000, B 0.000, C 0.000 }
gfCNCPoint3[13730] = {X 515.9212, Y 20.0113, Z -4.6667, A 0.000, B 0.000, C 0.000 }
gfCNCPoint3[13731] = {X 515.4650, Y 19.1639, Z -4.6667, A 0.000, B 0.000, C 0.000 }
gfCNCPoint3[13732] = {X 515.1840, Y 18.2434, Z -4.6667, A 0.000, B 0.000, C 0.000 }
gfCNCPoint3[13733] = {X 515.0891, Y 17.2857, Z -4.6667, A 0.000, B 0.000, C 0.000 }
gfCNCPoint3[13734] = {X 515.0891, Y 10.3077, Z -4.6667, A 0.000, B 0.000, C 0.000 }
gfCNCPoint3[13735] = {X 515.0966, Y 10.0382, Z -4.6667, A 0.000, B 0.000, C 0.000 }
gfCNCPoint3[13736] = {X 515.1189, Y 9.7696, Z -4.6667, A 0.000, B 0.000, C 0.000 }
gfCNCPoint3[13737] = {X 515.3251, Y 8.8084, Z -4.6667, A 0.000, B 0.000, C 0.000 }
gfCNCPoint3[13738] = {X 515.7199, Y 7.9080, Z -4.6667, A 0.000, B 0.000, C 0.000 }
gfCNCPoint3[13739] = {X 516.2871, Y 7.1050, Z -4.6667, A 0.000, B 0.000, C 0.000 }
gfCNCPoint3[13740] = {X 516.6493, Y 7.4200, Z -4.6667, A 0.000, B 0.000, C 0.000 }
gfCNCPoint3[13741] = {X 517.3373, Y 6.7815, Z -4.6667, A 0.000, B 0.000, C 0.000 }
gfCNCPoint3[13742] = {X 518.1451, Y 6.3036, Z -4.6667, A 0.000, B 0.000, C 0.000 }
gfCNCPoint3[13743] = {X 519.0359, Y 6.0078, Z -4.6667, A 0.000, B 0.000, C 0.000 }
gfCNCPoint3[13744] = {X 519.9692, Y 5.9077, Z -4.6667, A 0.000, B 0.000, C 0.000 }
gfCNCPoint3[13745] = {X 520.6509, Y 5.9079, Z -4.6667, A 0.000, B 0.000, C 0.000 }
gfCNCPoint3[13746] = {X 521.4833, Y 5.9951, Z -4.6667, A 0.000, B 0.000, C 0.000 }
gfCNCPoint3[13747] = {X 522.2841, Y 6.2383, Z -4.6667, A 0.000, B 0.000, C 0.000 }
gfCNCPoint3[13748] = {X 523.0244, Y 6.6288, Z -4.6667, A 0.000, B 0.000, C 0.000 }
gfCNCPoint3[13749] = {X 523.6774, Y 7.1524, Z -4.6667, A 0.000, B 0.000, C 0.000 }
gfCNCPoint3[13750] = {X 524.2194, Y 7.7901, Z -4.6667, A 0.000, B 0.000, C 0.000 }
gfCNCPoint3[13751] = {X 543.7489, Y 7.7906, Z -4.6667, A 0.000, B 0.000, C 0.000 }
gfCNCPoint3[13752] = {X 544.7471, Y 7.8779, Z -4.6667, A 0.000, B 0.000, C 0.000 }
gfCNCPoint3[13753] = {X 545.6997, Y 8.1885, Z -4.6667, A 0.000, B 0.000, C 0.000 }
gfCNCPoint3[13754] = {X 546.5574, Y 8.7064, Z -4.6667, A 0.000, B 0.000, C 0.000 }
gfCNCPoint3[13755] = {X 547.2760, Y 9.4048, Z -4.6667, A 0.000, B 0.000, C 0.000 }
gfCNCPoint3[13756] = {X 547.8181, Y 10.2475, Z -4.6667, A 0.000, B 0.000, C 0.000 }
gfCNCPoint3[13757] = {X 548.1557, Y 11.1909, Z -4.6667, A 0.000, B 0.000, C 0.000 }
gfCNCPoint3[13758] = {X 548.2714, Y 12.1862, Z -4.6667, A 0.000, B 0.000, C 0.000 }
gfCNCPoint3[13759] = {X 548.2712, Y 13.0233, Z -4.6667, A 0.000, B 0.000, C 0.000 }
gfCNCPoint3[13760] = {X 548.1629, Y 13.9494, Z -4.6667, A 0.000, B 0.000, C 0.000 }
gfCNCPoint3[13761] = {X 547.8618, Y 14.8318, Z -4.6667, A 0.000, B 0.000, C 0.000 }
gfCNCPoint3[13762] = {X 547.3816, Y 15.6310, Z -4.6667, A 0.000, B 0.000, C 0.000 }
gfCNCPoint3[13763] = {X 546.7438, Y 16.3111, Z -4.6667, A 0.000, B 0.000, C 0.000 }
gfCNCPoint3[13764] = {X 546.7440, Y 40.8759, Z -4.6667, A 0.000, B 0.000, C 0.000 }
gfCNCPoint3[13765] = {X 547.3886, Y 41.5650, Z -4.6667, A 0.000, B 0.000, C 0.000 }
gfCNCPoint3[13766] = {X 547.8714, Y 42.3757, Z -4.6667, A 0.000, B 0.000, C 0.000 }
gfCNCPoint3[13767] = {X 548.1703, Y 43.2707, Z -4.6667, A 0.000, B 0.000, C 0.000 }
gfCNCPoint3[13768] = {X 548.2714, Y 44.2089, Z -4.6667, A 0.000, B 0.000, C 0.000 }
gfCNCPoint3[13769] = {X 548.2714, Y 45.0006, Z -4.6667, A 0.000, B 0.000, C 0.000 }
gfCNCPoint3[13770] = {X 548.1558, Y 45.9959, Z -4.6667, A 0.000, B 0.000, C 0.000 }
gfCNCPoint3[13771] = {X 547.8181, Y 46.9393, Z -4.6667, A 0.000, B 0.000, C 0.000 }
gfCNCPoint3[13772] = {X 547.2760, Y 47.7820, Z -4.6667, A 0.000, B 0.000, C 0.000 }
gfCNCPoint3[13773] = {X 546.5575, Y 48.4803, Z -4.6667, A 0.000, B 0.000, C 0.000 }
gfCNCPoint3[13774] = {X 545.6997, Y 48.9981, Z -4.6667, A 0.000, B 0.000, C 0.000 }
gfCNCPoint3[13775] = {X 544.7470, Y 49.3087, Z -4.6667, A 0.000, B 0.000, C 0.000 }
gfCNCPoint3[13776] = {X 543.7488, Y 49.3959, Z -4.6667, A 0.000, B 0.000, C 0.000 }
gfCNCPoint3[13777] = {X 524.0862, Y 49.3964, Z -4.6667, A 0.000, B 0.000, C 0.000 }
gfCNCPoint3[13778] = {X 523.5294, Y 50.0314, Z -4.6667, A 0.000, B 0.000, C 0.000 }
gfCNCPoint3[13779] = {X 522.8651, Y 50.5528, Z -4.6667, A 0.000, B 0.000, C 0.000 }
gfCNCPoint3[13780] = {X 522.1159, Y 50.9426, Z -4.6667, A 0.000, B 0.000, C 0.000 }
gfCNCPoint3[13781] = {X 521.3077, Y 51.1875, Z -4.6667, A 0.000, B 0.000, C 0.000 }
gfCNCPoint3[13782] = {X 520.4681, Y 51.2791, Z -4.6667, A 0.000, B 0.000, C 0.000 }
gfCNCPoint3[13783] = {X 519.7998, Y 51.2791, Z -4.6667, A 0.000, B 0.000, C 0.000 }
gfCNCPoint3[13784] = {X 518.8207, Y 51.1688, Z -4.6667, A 0.000, B 0.000, C 0.000 }
gfCNCPoint3[13785] = {X 517.8907, Y 50.8434, Z -4.6667, A 0.000, B 0.000, C 0.000 }
gfCNCPoint3[13786] = {X 517.0564, Y 50.3192, Z -4.6667, A 0.000, B 0.000, C 0.000 }
gfCNCPoint3[13787] = {X 516.3597, Y 49.6225, Z -4.6667, A 0.000, B 0.000, C 0.000 }
gfCNCPoint3[13788] = {X 515.8355, Y 48.7882, Z -4.6667, A 0.000, B 0.000, C 0.000 }
gfCNCPoint3[13789] = {X 515.5101, Y 47.8582, Z -4.6667, A 0.000, B 0.000, C 0.000 }
gfCNCPoint3[13790] = {X 515.3998, Y 46.8791, Z -4.6667, A 0.000, B 0.000, C 0.000 }
gfCNCPoint3[13791] = {X 515.3998, Y 39.9011, Z -4.6667, A 0.000, B 0.000, C 0.000 }
gfCNCPoint3[13792] = {X 515.5101, Y 38.9220, Z -4.6667, A 0.000, B 0.000, C 0.000 }
gfCNCPoint3[13793] = {X 515.8355, Y 37.9920, Z -4.6667, A 0.000, B 0.000, C 0.000 }
gfCNCPoint3[13794] = {X 516.3597, Y 37.1577, Z -4.6667, A 0.000, B 0.000, C 0.000 }
gfCNCPoint3[13795] = {X 517.0565, Y 36.4610, Z -4.6667, A 0.000, B 0.000, C 0.000 }
gfCNCPoint3[13796] = {X 517.8907, Y 35.9368, Z -4.6667, A 0.000, B 0.000, C 0.000 }
gfCNCPoint3[13797] = {X 518.8207, Y 35.6114, Z -4.6667, A 0.000, B 0.000, C 0.000 }
gfCNCPoint3[13798] = {X 519.7998, Y 35.5011, Z -4.6667, A 0.000, B 0.000, C 0.000 }
gfCNCPoint3[13799] = {X 520.5280, Y 35.5015, Z -4.6667, A 0.000, B 0.000, C 0.000 }
gfCNCPoint3[13800] = {X 521.3614, Y 35.5927, Z -4.6667, A 0.000, B 0.000, C 0.000 }
gfCNCPoint3[13801] = {X 522.1624, Y 35.8403, Z -4.6667, A 0.000, B 0.000, C 0.000 }
gfCNCPoint3[13802] = {X 522.9018, Y 36.2354, Z -4.6667, A 0.000, B 0.000, C 0.000 }
gfCNCPoint3[13803] = {X 523.5529, Y 36.7635, Z -4.6667, A 0.000, B 0.000, C 0.000 }
gfCNCPoint3[13804] = {X 524.0921, Y 37.4056, Z -4.6667, A 0.000, B 0.000, C 0.000 }
gfCNCPoint3[13805] = {X 534.5519, Y 37.4061, Z -4.6667, A 0.000, B 0.000, C 0.000 }
gfCNCPoint3[13806] = {X 534.5519, Y 34.0455, Z -4.6667, A 0.000, B 0.000, C 0.000 }
gfCNCPoint3[13807] = {X 530.1522, Y 34.0451, Z -4.6667, A 0.000, B 0.000, C 0.000 }
gfCNCPoint3[13808] = {X 529.6045, Y 34.6955, Z -4.6667, A 0.000, B 0.000, C 0.000 }
gfCNCPoint3[13809] = {X 528.9420, Y 35.2284, Z -4.6667, A 0.000, B 0.000, C 0.000 }
gfCNCPoint3[13810] = {X 528.1893, Y 35.6239, Z -4.6667, A 0.000, B 0.000, C 0.000 }
gfCNCPoint3[13811] = {X 527.3746, Y 35.8673, Z -4.6667, A 0.000, B 0.000, C 0.000 }
gfCNCPoint3[13812] = {X 526.5283, Y 35.9495, Z -4.6667, A 0.000, B 0.000, C 0.000 }
gfCNCPoint3[13813] = {X 525.8868, Y 35.9495, Z -4.6667, A 0.000, B 0.000, C 0.000 }
gfCNCPoint3[13814] = {X 524.9077, Y 35.8391, Z -4.6667, A 0.000, B 0.000, C 0.000 }
gfCNCPoint3[13815] = {X 523.9777, Y 35.5137, Z -4.6667, A 0.000, B 0.000, C 0.000 }
gfCNCPoint3[13816] = {X 523.1434, Y 34.9895, Z -4.6667, A 0.000, B 0.000, C 0.000 }
gfCNCPoint3[13817] = {X 522.4467, Y 34.2928, Z -4.6667, A 0.000, B 0.000, C 0.000 }
gfCNCPoint3[13818] = {X 521.9225, Y 33.4585, Z -4.6667, A 0.000, B 0.000, C 0.000 }
gfCNCPoint3[13819] = {X 521.5971, Y 32.5285, Z -4.6667, A 0.000, B 0.000, C 0.000 }
gfCNCPoint3[13820] = {X 521.4868, Y 31.5495, Z -4.6667, A 0.000, B 0.000, C 0.000 }
gfCNCPoint3[13821] = {X 521.4868, Y 24.5714, Z -4.6667, A 0.000, B 0.000, C 0.000 }
gfCNCPoint3[13822] = {X 521.5971, Y 23.5923, Z -4.6667, A 0.000, B 0.000, C 0.000 }
gfCNCPoint3[13823] = {X 521.9225, Y 22.6623, Z -4.6667, A 0.000, B 0.000, C 0.000 }
gfCNCPoint3[13824] = {X 522.4467, Y 21.8281, Z -4.6667, A 0.000, B 0.000, C 0.000 }
gfCNCPoint3[13825] = {X 523.1434, Y 21.1314, Z -4.6667, A 0.000, B 0.000, C 0.000 }
gfCNCPoint3[13826] = {X 523.9777, Y 20.6072, Z -4.6667, A 0.000, B 0.000, C 0.000 }
gfCNCPoint3[13827] = {X 524.9077, Y 20.2817, Z -4.6667, A 0.000, B 0.000, C 0.000 }
gfCNCPoint3[13828] = {X 525.8868, Y 20.1714, Z -4.6667, A 0.000, B 0.000, C 0.000 }
gfCNCPoint3[13829] = {X 526.5702, Y 20.1716, Z -4.6667, A 0.000, B 0.000, C 0.000 }
gfCNCPoint3[13830] = {X 527.4023, Y 20.2591, Z -4.6667, A 0.000, B 0.000, C 0.000 }
gfCNCPoint3[13831] = {X 528.2027, Y 20.5024, Z -4.6667, A 0.000, B 0.000, C 0.000 }
gfCNCPoint3[13832] = {X 528.9426, Y 20.8929, Z -4.6667, A 0.000, B 0.000, C 0.000 }
gfCNCPoint3[13833] = {X 529.5952, Y 21.4163, Z -4.6667, A 0.000, B 0.000, C 0.000 }
gfCNCPoint3[13834] = {X 530.1370, Y 22.0538, Z -4.6667, A 0.000, B 0.000, C 0.000 }
gfCNCPoint3[13835] = {X 534.5519, Y 22.0541, Z -4.6667, A 0.000, B 0.000, C 0.000 }
gfCNCPoint3[13836] = {X 534.5519, Y 19.7819, Z -4.6667, A 0.000, B 0.000, C 0.000 }
gfCNCPoint3[13837] = {X 528.8177, Y 19.7817, Z -4.6667, A 0.000, B 0.000, C 0.000 }
gfCNCPoint3[13838] = {X 528.8177, Y 20.2617, Z -4.6667, A 0.000, B 0.000, C 0.000 }
gfCNCPoint3[13839] = {X 534.0719, Y 20.2619, Z -4.6667, A 0.000, B 0.000, C 0.000 }
gfCNCPoint3[13840] = {X 534.0719, Y 21.5740, Z -4.6667, A 0.000, B 0.000, C 0.000 }
gfCNCPoint3[13841] = {X 530.3792, Y 21.5738, Z -4.6667, A 0.000, B 0.000, C 0.000 }
gfCNCPoint3[13842] = {X 529.6678, Y 20.8353, Z -4.6667, A 0.000, B 0.000, C 0.000 }
gfCNCPoint3[13843] = {X 528.8177, Y 20.2617, Z -4.6667, A 0.000, B 0.000, C 0.000 }
gfCNCPoint3[13844] = {X 528.8177, Y 19.7817, Z -4.6667, A 0.000, B 0.000, C 0.000 }
gfCNCPoint3[13845] = {X 524.2344, Y 19.7816, Z -4.6667, A 0.000, B 0.000, C 0.000 }
gfCNCPoint3[13846] = {X 523.6867, Y 20.4319, Z -4.6667, A 0.000, B 0.000, C 0.000 }
gfCNCPoint3[13847] = {X 523.0242, Y 20.9648, Z -4.6667, A 0.000, B 0.000, C 0.000 }
gfCNCPoint3[13848] = {X 522.2716, Y 21.3602, Z -4.6667, A 0.000, B 0.000, C 0.000 }
gfCNCPoint3[13849] = {X 521.4569, Y 21.6036, Z -4.6667, A 0.000, B 0.000, C 0.000 }
gfCNCPoint3[13850] = {X 520.6107, Y 21.6857, Z -4.6667, A 0.000, B 0.000, C 0.000 }
gfCNCPoint3[13851] = {X 519.9691, Y 21.6857, Z -4.6667, A 0.000, B 0.000, C 0.000 }
gfCNCPoint3[13852] = {X 518.9900, Y 21.5754, Z -4.6667, A 0.000, B 0.000, C 0.000 }
gfCNCPoint3[13853] = {X 518.0600, Y 21.2500, Z -4.6667, A 0.000, B 0.000, C 0.000 }
gfCNCPoint3[13854] = {X 517.2257, Y 20.7258, Z -4.6667, A 0.000, B 0.000, C 0.000 }
gfCNCPoint3[13855] = {X 516.5290, Y 20.0291, Z -4.6667, A 0.000, B 0.000, C 0.000 }
gfCNCPoint3[13856] = {X 516.0048, Y 19.1948, Z -4.6667, A 0.000, B 0.000, C 0.000 }
gfCNCPoint3[13857] = {X 515.6794, Y 18.2648, Z -4.6667, A 0.000, B 0.000, C 0.000 }
gfCNCPoint3[13858] = {X 515.5691, Y 17.2857, Z -4.6667, A 0.000, B 0.000, C 0.000 }
gfCNCPoint3[13859] = {X 515.5691, Y 10.3077, Z -4.6667, A 0.000, B 0.000, C 0.000 }
gfCNCPoint3[13860] = {X 515.6394, Y 9.5244, Z -4.6667, A 0.000, B 0.000, C 0.000 }
gfCNCPoint3[13861] = {X 515.8480, Y 8.7661, Z -4.6667, A 0.000, B 0.000, C 0.000 }
gfCNCPoint3[13862] = {X 516.1882, Y 8.0571, Z -4.6667, A 0.000, B 0.000, C 0.000 }
gfCNCPoint3[13863] = {X 516.6493, Y 7.4200, Z -4.6667, A 0.000, B 0.000, C 0.000 }
gfCNCPoint3[13864] = {X 516.2871, Y 7.1050, Z -4.6667, A 0.000, B 0.000, C 0.000 }
gfCNCPoint3[13865] = {X 469.2605, Y 7.1050, Z -4.6667, A 0.000, B 0.000, C 0.000 }
gfCNCPoint3[13866] = {X 469.2605, Y 11.9050, Z -4.6667, A 0.000, B 0.000, C 0.000 }
gfCNCPoint3[13867] = {X 469.1140, Y 11.9050, Z -4.6667, A 0.000, B 0.000, C 0.000 }
gfCNCPoint3[13868] = {X 469.1170, Y 12.0436, Z -4.6667, A 0.000, B 0.000, C 0.000 }
gfCNCPoint3[13869] = {X 469.1179, Y 12.1822, Z -4.6667, A 0.000, B 0.000, C 0.000 }
gfCNCPoint3[13870] = {X 469.1886, Y 12.0433, Z -4.6667, A 0.000, B 0.000, C 0.000 }
gfCNCPoint3[13871] = {X 469.2605, Y 11.9050, Z -4.6667, A 0.000, B 0.000, C 0.000 }
gfCNCPoint3[13872] = {X 469.2605, Y 9.5050, Z -4.6667, A 0.000, B 0.000, C 0.000 }
gfCNCPoint3[13873] = {X 466.2073, Y 9.5050, Z -4.6667, A 0.000, B 0.000, C 0.000 }
gfCNCPoint3[13874] = {X 466.5689, Y 10.7172, Z -4.6667, A 0.000, B 0.000, C 0.000 }
gfCNCPoint3[13875] = {X 466.7150, Y 11.9737, Z -4.6667, A 0.000, B 0.000, C 0.000 }
gfCNCPoint3[13876] = {X 466.7172, Y 12.0777, Z -4.6667, A 0.000, B 0.000, C 0.000 }
gfCNCPoint3[13877] = {X 466.7179, Y 12.1818, Z -4.6667, A 0.000, B 0.000, C 0.000 }
gfCNCPoint3[13878] = {X 466.7179, Y 12.9779, Z -4.6667, A 0.000, B 0.000, C 0.000 }
gfCNCPoint3[13879] = {X 466.6191, Y 14.1733, Z -4.6667, A 0.000, B 0.000, C 0.000 }
gfCNCPoint3[13880] = {X 466.3254, Y 15.3363, Z -4.6667, A 0.000, B 0.000, C 0.000 }
gfCNCPoint3[13881] = {X 465.8447, Y 16.4352, Z -4.6667, A 0.000, B 0.000, C 0.000 }
gfCNCPoint3[13882] = {X 465.1900, Y 17.4403, Z -4.6667, A 0.000, B 0.000, C 0.000 }
gfCNCPoint3[13883] = {X 465.1904, Y 25.8784, Z -4.6667, A 0.000, B 0.000, C 0.000 }
gfCNCPoint3[13884] = {X 467.5904, Y 25.8783, Z -4.6667, A 0.000, B 0.000, C 0.000 }
gfCNCPoint3[13885] = {X 467.5910, Y 38.9905, Z -4.6667, A 0.000, B 0.000, C 0.000 }
gfCNCPoint3[13886] = {X 467.6015, Y 39.0069, Z -4.6667, A 0.000, B 0.000, C 0.000 }
gfCNCPoint3[13887] = {X 468.3506, Y 37.9855, Z -4.6667, A 0.000, B 0.000, C 0.000 }
gfCNCPoint3[13888] = {X 469.2267, Y 37.0706, Z -4.6667, A 0.000, B 0.000, C 0.000 }
gfCNCPoint3[13889] = {X 470.2148, Y 36.2780, Z -4.6667, A 0.000, B 0.000, C 0.000 }
gfCNCPoint3[13890] = {X 471.5278, Y 33.7079, Z -4.6667, A 0.000, B 0.000, C 0.000 }
gfCNCPoint3[13891] = {X 470.4809, Y 32.4120, Z -4.6667, A 0.000, B 0.000, C 0.000 }
gfCNCPoint3[13892] = {X 469.5673, Y 31.0190, Z -4.6667, A 0.000, B 0.000, C 0.000 }
gfCNCPoint3[13893] = {X 468.7959, Y 29.5425, Z -4.6667, A 0.000, B 0.000, C 0.000 }
gfCNCPoint3[13894] = {X 468.1742, Y 27.9969, Z -4.6667, A 0.000, B 0.000, C 0.000 }
gfCNCPoint3[13895] = {X 467.7084, Y 26.3975, Z -4.6667, A 0.000, B 0.000, C 0.000 }
gfCNCPoint3[13896] = {X 467.6478, Y 26.1382, Z -4.6667, A 0.000, B 0.000, C 0.000 }
gfCNCPoint3[13897] = {X 467.5904, Y 25.8783, Z -4.6667, A 0.000, B 0.000, C 0.000 }
gfCNCPoint3[13898] = {X 465.1904, Y 25.8784, Z -4.6667, A 0.000, B 0.000, C 0.000 }
gfCNCPoint3[13899] = {X 465.1910, Y 39.7478, Z -4.6667, A 0.000, B 0.000, C 0.000 }
gfCNCPoint3[13900] = {X 465.3905, Y 40.0177, Z -4.6667, A 0.000, B 0.000, C 0.000 }
gfCNCPoint3[13901] = {X 465.5774, Y 40.2966, Z -4.6667, A 0.000, B 0.000, C 0.000 }
gfCNCPoint3[13902] = {X 466.0634, Y 41.1919, Z -4.6667, A 0.000, B 0.000, C 0.000 }
gfCNCPoint3[13903] = {X 466.4196, Y 42.1462, Z -4.6667, A 0.000, B 0.000, C 0.000 }
gfCNCPoint3[13904] = {X 466.6392, Y 43.1408, Z -4.6667, A 0.000, B 0.000, C 0.000 }
gfCNCPoint3[13905] = {X 466.7178, Y 44.1564, Z -4.6667, A 0.000, B 0.000, C 0.000 }
gfCNCPoint3[13906] = {X 466.7179, Y 45.0000, Z -4.6667, A 0.000, B 0.000, C 0.000 }
gfCNCPoint3[13907] = {X 466.7033, Y 45.4609, Z -4.6667, A 0.000, B 0.000, C 0.000 }
gfCNCPoint3[13908] = {X 466.6596, Y 45.9200, Z -4.6667, A 0.000, B 0.000, C 0.000 }
gfCNCPoint3[13909] = {X 468.5433, Y 45.9200, Z -4.6667, A 0.000, B 0.000, C 0.000 }
gfCNCPoint3[13910] = {X 468.4996, Y 45.4609, Z -4.6667, A 0.000, B 0.000, C 0.000 }
gfCNCPoint3[13911] = {X 468.4850, Y 45.0000, Z -4.6667, A 0.000, B 0.000, C 0.000 }
gfCNCPoint3[13912] = {X 468.4850, Y 44.2089, Z -4.6667, A 0.000, B 0.000, C 0.000 }
gfCNCPoint3[13913] = {X 468.5580, Y 43.1798, Z -4.6667, A 0.000, B 0.000, C 0.000 }
gfCNCPoint3[13914] = {X 468.7759, Y 42.1714, Z -4.6667, A 0.000, B 0.000, C 0.000 }
gfCNCPoint3[13915] = {X 469.1341, Y 41.2038, Z -4.6667, A 0.000, B 0.000, C 0.000 }
gfCNCPoint3[13916] = {X 469.6255, Y 40.2966, Z -4.6667, A 0.000, B 0.000, C 0.000 }
gfCNCPoint3[13917] = {X 470.3102, Y 39.3876, Z -4.6667, A 0.000, B 0.000, C 0.000 }
gfCNCPoint3[13918] = {X 471.1282, Y 38.5964, Z -4.6667, A 0.000, B 0.000, C 0.000 }
gfCNCPoint3[13919] = {X 472.0595, Y 37.9424, Z -4.6667, A 0.000, B 0.000, C 0.000 }
gfCNCPoint3[13920] = {X 474.4570, Y 33.2495, Z -4.6667, A 0.000, B 0.000, C 0.000 }
gfCNCPoint3[13921] = {X 473.2256, Y 32.0050, Z -4.6667, A 0.000, B 0.000, C 0.000 }
gfCNCPoint3[13922] = {X 472.1540, Y 30.6204, Z -4.6667, A 0.000, B 0.000, C 0.000 }
gfCNCPoint3[13923] = {X 471.2580, Y 29.1163, Z -4.6667, A 0.000, B 0.000, C 0.000 }
gfCNCPoint3[13924] = {X 470.5507, Y 27.5148, Z -4.6667, A 0.000, B 0.000, C 0.000 }
gfCNCPoint3[13925] = {X 470.0426, Y 25.8393, Z -4.6667, A 0.000, B 0.000, C 0.000 }
gfCNCPoint3[13926] = {X 469.9883, Y 25.6073, Z -4.6667, A 0.000, B 0.000, C 0.000 }
gfCNCPoint3[13927] = {X 469.9369, Y 25.3747, Z -4.6667, A 0.000, B 0.000, C 0.000 }
gfCNCPoint3[13928] = {X 469.6261, Y 23.4808, Z -4.6667, A 0.000, B 0.000, C 0.000 }
gfCNCPoint3[13929] = {X 469.5013, Y 21.5656, Z -4.6667, A 0.000, B 0.000, C 0.000 }
gfCNCPoint3[13930] = {X 469.5635, Y 19.6474, Z -4.6667, A 0.000, B 0.000, C 0.000 }
gfCNCPoint3[13931] = {X 469.8123, Y 17.7443, Z -4.6667, A 0.000, B 0.000, C 0.000 }
gfCNCPoint3[13932] = {X 470.2453, Y 15.8746, Z -4.6667, A 0.000, B 0.000, C 0.000 }
gfCNCPoint3[13933] = {X 470.6916, Y 14.5433, Z -4.6667, A 0.000, B 0.000, C 0.000 }
gfCNCPoint3[13934] = {X 471.2621, Y 13.2604, Z -4.6667, A 0.000, B 0.000, C 0.000 }
gfCNCPoint3[13935] = {X 471.3229, Y 13.1409, Z -4.6667, A 0.000, B 0.000, C 0.000 }
gfCNCPoint3[13936] = {X 471.3848, Y 13.0219, Z -4.6667, A 0.000, B 0.000, C 0.000 }
gfCNCPoint3[13937] = {X 472.1259, Y 11.7667, Z -4.6667, A 0.000, B 0.000, C 0.000 }
gfCNCPoint3[13938] = {X 472.9869, Y 10.5906, Z -4.6667, A 0.000, B 0.000, C 0.000 }
gfCNCPoint3[13939] = {X 473.9595, Y 9.5050, Z -4.6667, A 0.000, B 0.000, C 0.000 }
gfCNCPoint3[13940] = {X 469.2605, Y 9.5050, Z -4.6667, A 0.000, B 0.000, C 0.000 }
gfCNCPoint3[13941] = {X 469.2605, Y 7.1050, Z -4.6667, A 0.000, B 0.000, C 0.000 }
gfCNCPoint3[13942] = {X 370.1027, Y 7.1050, Z -4.6667, A 0.000, B 0.000, C 0.000 }
gfCNCPoint3[13943] = {X 371.1262, Y 8.7919, Z -4.6667, A 0.000, B 0.000, C 0.000 }
gfCNCPoint3[13944] = {X 372.0369, Y 10.5423, Z -4.6667, A 0.000, B 0.000, C 0.000 }
gfCNCPoint3[13945] = {X 372.9282, Y 12.5944, Z -4.6667, A 0.000, B 0.000, C 0.000 }
gfCNCPoint3[13946] = {X 373.6645, Y 14.7071, Z -4.6667, A 0.000, B 0.000, C 0.000 }
gfCNCPoint3[13947] = {X 374.2417, Y 16.8687, Z -4.6667, A 0.000, B 0.000, C 0.000 }
gfCNCPoint3[13948] = {X 374.7312, Y 19.4365, Z -4.6667, A 0.000, B 0.000, C 0.000 }
gfCNCPoint3[13949] = {X 375.0380, Y 22.0324, Z -4.6667, A 0.000, B 0.000, C 0.000 }
gfCNCPoint3[13950] = {X 375.1606, Y 24.6435, Z -4.6667, A 0.000, B 0.000, C 0.000 }
gfCNCPoint3[13951] = {X 375.0985, Y 27.2568, Z -4.6667, A 0.000, B 0.000, C 0.000 }
gfCNCPoint3[13952] = {X 374.8518, Y 29.8591, Z -4.6667, A 0.000, B 0.000, C 0.000 }
gfCNCPoint3[13953] = {X 374.4219, Y 32.4375, Z -4.6667, A 0.000, B 0.000, C 0.000 }
gfCNCPoint3[13954] = {X 373.7852, Y 34.9948, Z -4.6667, A 0.000, B 0.000, C 0.000 }
gfCNCPoint3[13955] = {X 372.9257, Y 37.4861, Z -4.6667, A 0.000, B 0.000, C 0.000 }
gfCNCPoint3[13956] = {X 371.8501, Y 39.8920, Z -4.6667, A 0.000, B 0.000, C 0.000 }
gfCNCPoint3[13957] = {X 370.5668, Y 42.1937, Z -4.6667, A 0.000, B 0.000, C 0.000 }
gfCNCPoint3[13958] = {X 369.0856, Y 44.3735, Z -4.6667, A 0.000, B 0.000, C 0.000 }
gfCNCPoint3[13959] = {X 368.9519, Y 44.5568, Z -4.6667, A 0.000, B 0.000, C 0.000 }
gfCNCPoint3[13960] = {X 368.8455, Y 44.6947, Z -4.6667, A 0.000, B 0.000, C 0.000 }
gfCNCPoint3[13961] = {X 368.1809, Y 45.5108, Z -4.6667, A 0.000, B 0.000, C 0.000 }
gfCNCPoint3[13962] = {X 366.6024, Y 47.2819, Z -4.6667, A 0.000, B 0.000, C 0.000 }
gfCNCPoint3[13963] = {X 364.8727, Y 48.9057, Z -4.6667, A 0.000, B 0.000, C 0.000 }
gfCNCPoint3[13964] = {X 363.0054, Y 50.3692, Z -4.6667, A 0.000, B 0.000, C 0.000 }
gfCNCPoint3[13965] = {X 361.0155, Y 51.6610, Z -4.6667, A 0.000, B 0.000, C 0.000 }
gfCNCPoint3[13966] = {X 358.9186, Y 52.7707, Z -4.6667, A 0.000, B 0.000, C 0.000 }
gfCNCPoint3[13967] = {X 358.3784, Y 53.0236, Z -4.6667, A 0.000, B 0.000, C 0.000 }
gfCNCPoint3[13968] = {X 356.2272, Y 53.8549, Z -4.6667, A 0.000, B 0.000, C 0.000 }
gfCNCPoint3[13969] = {X 354.0156, Y 54.5088, Z -4.6667, A 0.000, B 0.000, C 0.000 }
gfCNCPoint3[13970] = {X 351.7583, Y 54.9809, Z -4.6667, A 0.000, B 0.000, C 0.000 }
gfCNCPoint3[13971] = {X 349.4700, Y 55.2682, Z -4.6667, A 0.000, B 0.000, C 0.000 }
gfCNCPoint3[13972] = {X 347.1660, Y 55.3688, Z -4.6667, A 0.000, B 0.000, C 0.000 }
gfCNCPoint3[13973] = {X 344.5859, Y 55.3170, Z -4.6667, A 0.000, B 0.000, C 0.000 }
gfCNCPoint3[13974] = {X 342.0205, Y 55.0374, Z -4.6667, A 0.000, B 0.000, C 0.000 }
gfCNCPoint3[13975] = {X 339.4899, Y 54.5321, Z -4.6667, A 0.000, B 0.000, C 0.000 }
gfCNCPoint3[13976] = {X 337.0138, Y 53.8051, Z -4.6667, A 0.000, B 0.000, C 0.000 }
gfCNCPoint3[13977] = {X 334.7576, Y 52.9264, Z -4.6667, A 0.000, B 0.000, C 0.000 }
gfCNCPoint3[13978] = {X 332.5820, Y 51.8637, Z -4.6667, A 0.000, B 0.000, C 0.000 }
gfCNCPoint3[13979] = {X 331.5868, Y 51.2788, Z -4.6667, A 0.000, B 0.000, C 0.000 }
gfCNCPoint3[13980] = {X 330.6155, Y 50.6549, Z -4.6667, A 0.000, B 0.000, C 0.000 }
gfCNCPoint3[13981] = {X 331.5807, Y 51.6087, Z -4.6667, A 0.000, B 0.000, C 0.000 }
gfCNCPoint3[13982] = {X 332.4030, Y 52.6881, Z -4.6667, A 0.000, B 0.000, C 0.000 }
gfCNCPoint3[13983] = {X 333.0663, Y 53.8719, Z -4.6667, A 0.000, B 0.000, C 0.000 }
gfCNCPoint3[13984] = {X 333.5576, Y 55.1368, Z -4.6667, A 0.000, B 0.000, C 0.000 }
gfCNCPoint3[13985] = {X 333.8671, Y 56.4580, Z -4.6667, A 0.000, B 0.000, C 0.000 }
gfCNCPoint3[13986] = {X 333.9597, Y 57.2265, Z -4.6667, A 0.000, B 0.000, C 0.000 }
gfCNCPoint3[13987] = {X 333.9907, Y 58.0000, Z -4.6667, A 0.000, B 0.000, C 0.000 }
gfCNCPoint3[13988] = {X 333.9907, Y 58.9444, Z -4.6667, A 0.000, B 0.000, C 0.000 }
gfCNCPoint3[13989] = {X 333.8761, Y 60.3996, Z -4.6667, A 0.000, B 0.000, C 0.000 }
gfCNCPoint3[13990] = {X 333.5448, Y 61.8211, Z -4.6667, A 0.000, B 0.000, C 0.000 }
gfCNCPoint3[13991] = {X 333.0044, Y 63.1770, Z -4.6667, A 0.000, B 0.000, C 0.000 }
gfCNCPoint3[13992] = {X 332.2670, Y 64.4367, Z -4.6667, A 0.000, B 0.000, C 0.000 }
gfCNCPoint3[13993] = {X 331.3492, Y 65.5717, Z -4.6667, A 0.000, B 0.000, C 0.000 }
gfCNCPoint3[13994] = {X 330.2718, Y 66.5565, Z -4.6667, A 0.000, B 0.000, C 0.000 }
gfCNCPoint3[13995] = {X 330.2732, Y 83.2031, Z -4.6667, A 0.000, B 0.000, C 0.000 }
gfCNCPoint3[13996] = {X 330.2770, Y 83.5829, Z -4.6667, A 0.000, B 0.000, C 0.000 }
gfCNCPoint3[13997] = {X 330.3835, Y 83.6082, Z -4.6667, A 0.000, B 0.000, C 0.000 }
gfCNCPoint3[13998] = {X 333.0882, Y 84.1506, Z -4.6667, A 0.000, B 0.000, C 0.000 }
gfCNCPoint3[13999] = {X 335.8250, Y 84.4964, Z -4.6667, A 0.000, B 0.000, C 0.000 }
gfCNCPoint3[14000] = {X 339.8030, Y 84.8044, Z -4.6667, A 0.000, B 0.000, C 0.000 }
gfCNCPoint3[14001] = {X 343.7892, Y 84.9768, Z -4.6667, A 0.000, B 0.000, C 0.000 }
gfCNCPoint3[14002] = {X 347.7789, Y 85.0132, Z -4.6667, A 0.000, B 0.000, C 0.000 }
gfCNCPoint3[14003] = {X 351.9889, Y 84.9778, Z -4.6667, A 0.000, B 0.000, C 0.000 }
gfCNCPoint3[14004] = {X 356.1949, Y 84.7902, Z -4.6667, A 0.000, B 0.000, C 0.000 }
gfCNCPoint3[14005] = {X 360.3914, Y 84.4509, Z -4.6667, A 0.000, B 0.000, C 0.000 }
gfCNCPoint3[14006] = {X 362.9934, Y 84.1041, Z -4.6667, A 0.000, B 0.000, C 0.000 }
gfCNCPoint3[14007] = {X 365.5601, Y 83.5541, Z -4.6667, A 0.000, B 0.000, C 0.000 }
gfCNCPoint3[14008] = {X 365.5589, Y 66.5614, Z -4.6667, A 0.000, B 0.000, C 0.000 }
gfCNCPoint3[14009] = {X 364.4965, Y 65.5961, Z -4.6667, A 0.000, B 0.000, C 0.000 }
gfCNCPoint3[14010] = {X 363.5885, Y 64.4843, Z -4.6667, A 0.000, B 0.000, C 0.000 }
gfCNCPoint3[14011] = {X 362.8549, Y 63.2505, Z -4.6667, A 0.000, B 0.000, C 0.000 }
gfCNCPoint3[14012] = {X 349.9658, Y 69.6716, Z -4.6667, A 0.000, B 0.000, C 0.000 }
gfCNCPoint3[14013] = {X 348.6646, Y 69.7396, Z -4.6667, A 0.000, B 0.000, C 0.000 }
gfCNCPoint3[14014] = {X 347.3620, Y 69.7680, Z -4.6667, A 0.000, B 0.000, C 0.000 }
gfCNCPoint3[14015] = {X 346.5843, Y 69.7771, Z -4.6667, A 0.000, B 0.000, C 0.000 }
gfCNCPoint3[14016] = {X 345.8067, Y 69.7724, Z -4.6667, A 0.000, B 0.000, C 0.000 }
gfCNCPoint3[14017] = {X 345.5902, Y 70.1914, Z -4.6667, A 0.000, B 0.000, C 0.000 }
gfCNCPoint3[14018] = {X 345.3655, Y 70.6061, Z -4.6667, A 0.000, B 0.000, C 0.000 }
gfCNCPoint3[14019] = {X 346.5784, Y 70.6165, Z -4.6667, A 0.000, B 0.000, C 0.000 }
gfCNCPoint3[14020] = {X 347.7914, Y 70.6126, Z -4.6667, A 0.000, B 0.000, C 0.000 }
gfCNCPoint3[14021] = {X 349.1245, Y 70.6184, Z -4.6667, A 0.000, B 0.000, C 0.000 }
gfCNCPoint3[14022] = {X 350.4576, Y 70.6068, Z -4.6667, A 0.000, B 0.000, C 0.000 }
gfCNCPoint3[14023] = {X 350.2066, Y 70.1419, Z -4.6667, A 0.000, B 0.000, C 0.000 }
gfCNCPoint3[14024] = {X 349.9658, Y 69.6716, Z -4.6667, A 0.000, B 0.000, C 0.000 }
gfCNCPoint3[14025] = {X 352.1140, Y 68.6014, Z -4.6667, A 0.000, B 0.000, C 0.000 }
gfCNCPoint3[14026] = {X 351.7678, Y 67.8729, Z -4.6667, A 0.000, B 0.000, C 0.000 }
gfCNCPoint3[14027] = {X 351.4490, Y 67.1320, Z -4.6667, A 0.000, B 0.000, C 0.000 }
gfCNCPoint3[14028] = {X 349.3922, Y 67.3027, Z -4.6667, A 0.000, B 0.000, C 0.000 }
gfCNCPoint3[14029] = {X 347.3293, Y 67.3682, Z -4.6667, A 0.000, B 0.000, C 0.000 }
gfCNCPoint3[14030] = {X 345.8125, Y 67.3722, Z -4.6667, A 0.000, B 0.000, C 0.000 }
gfCNCPoint3[14031] = {X 344.2966, Y 67.3204, Z -4.6667, A 0.000, B 0.000, C 0.000 }
gfCNCPoint3[14032] = {X 343.8104, Y 68.3954, Z -4.6667, A 0.000, B 0.000, C 0.000 }
gfCNCPoint3[14033] = {X 343.2666, Y 69.4424, Z -4.6667, A 0.000, B 0.000, C 0.000 }
gfCNCPoint3[14034] = {X 342.7871, Y 70.2640, Z -4.6667, A 0.000, B 0.000, C 0.000 }
gfCNCPoint3[14035] = {X 342.2722, Y 71.0639, Z -4.6667, A 0.000, B 0.000, C 0.000 }
gfCNCPoint3[14036] = {X 342.2724, Y 72.9170, Z -4.6667, A 0.000, B 0.000, C 0.000 }
gfCNCPoint3[14037] = {X 343.8012, Y 72.9726, Z -4.6667, A 0.000, B 0.000, C 0.000 }
gfCNCPoint3[14038] = {X 345.3308, Y 73.0059, Z -4.6667, A 0.000, B 0.000, C 0.000 }
gfCNCPoint3[14039] = {X 346.5600, Y 73.0165, Z -4.6667, A 0.000, B 0.000, C 0.000 }
gfCNCPoint3[14040] = {X 347.7893, Y 73.0127, Z -4.6667, A 0.000, B 0.000, C 0.000 }
gfCNCPoint3[14041] = {X 349.1417, Y 73.0184, Z -4.6667, A 0.000, B 0.000, C 0.000 }
gfCNCPoint3[14042] = {X 350.4942, Y 73.0065, Z -4.6667, A 0.000, B 0.000, C 0.000 }
gfCNCPoint3[14043] = {X 352.0271, Y 72.9719, Z -4.6667, A 0.000, B 0.000, C 0.000 }
gfCNCPoint3[14044] = {X 353.5593, Y 72.9149, Z -4.6667, A 0.000, B 0.000, C 0.000 }
gfCNCPoint3[14045] = {X 353.5592, Y 71.0773, Z -4.6667, A 0.000, B 0.000, C 0.000 }
gfCNCPoint3[14046] = {X 353.0399, Y 70.2714, Z -4.6667, A 0.000, B 0.000, C 0.000 }
gfCNCPoint3[14047] = {X 352.5568, Y 69.4434, Z -4.6667, A 0.000, B 0.000, C 0.000 }
gfCNCPoint3[14048] = {X 352.3308, Y 69.0248, Z -4.6667, A 0.000, B 0.000, C 0.000 }
gfCNCPoint3[14049] = {X 352.1140, Y 68.6014, Z -4.6667, A 0.000, B 0.000, C 0.000 }
gfCNCPoint3[14050] = {X 354.2622, Y 67.5312, Z -4.6667, A 0.000, B 0.000, C 0.000 }
gfCNCPoint3[14051] = {X 353.5961, Y 66.0389, Z -4.6667, A 0.000, B 0.000, C 0.000 }
gfCNCPoint3[14052] = {X 353.0588, Y 64.4956, Z -4.6667, A 0.000, B 0.000, C 0.000 }
gfCNCPoint3[14053] = {X 350.1867, Y 64.8418, Z -4.6667, A 0.000, B 0.000, C 0.000 }
gfCNCPoint3[14054] = {X 347.2966, Y 64.9683, Z -4.6667, A 0.000, B 0.000, C 0.000 }
gfCNCPoint3[14055] = {X 344.9826, Y 64.9491, Z -4.6667, A 0.000, B 0.000, C 0.000 }
gfCNCPoint3[14056] = {X 342.6739, Y 64.7919, Z -4.6667, A 0.000, B 0.000, C 0.000 }
gfCNCPoint3[14057] = {X 341.9391, Y 66.7267, Z -4.6667, A 0.000, B 0.000, C 0.000 }
gfCNCPoint3[14058] = {X 341.0016, Y 68.5718, Z -4.6667, A 0.000, B 0.000, C 0.000 }
gfCNCPoint3[14059] = {X 339.8722, Y 70.3060, Z -4.6667, A 0.000, B 0.000, C 0.000 }
gfCNCPoint3[14060] = {X 339.8726, Y 75.1900, Z -4.6667, A 0.000, B 0.000, C 0.000 }
gfCNCPoint3[14061] = {X 343.8278, Y 75.3743, Z -4.6667, A 0.000, B 0.000, C 0.000 }
gfCNCPoint3[14062] = {X 347.7872, Y 75.4128, Z -4.6667, A 0.000, B 0.000, C 0.000 }
gfCNCPoint3[14063] = {X 351.8755, Y 75.3773, Z -4.6667, A 0.000, B 0.000, C 0.000 }
gfCNCPoint3[14064] = {X 355.9595, Y 75.1855, Z -4.6667, A 0.000, B 0.000, C 0.000 }
gfCNCPoint3[14065] = {X 355.9591, Y 70.3183, Z -4.6667, A 0.000, B 0.000, C 0.000 }
gfCNCPoint3[14066] = {X 355.0516, Y 68.9607, Z -4.6667, A 0.000, B 0.000, C 0.000 }
gfCNCPoint3[14067] = {X 354.2622, Y 67.5312, Z -4.6667, A 0.000, B 0.000, C 0.000 }
gfCNCPoint3[14068] = {X 356.4104, Y 66.4610, Z -4.6667, A 0.000, B 0.000, C 0.000 }
gfCNCPoint3[14069] = {X 355.7400, Y 64.9297, Z -4.6667, A 0.000, B 0.000, C 0.000 }
gfCNCPoint3[14070] = {X 355.2243, Y 63.3396, Z -4.6667, A 0.000, B 0.000, C 0.000 }
gfCNCPoint3[14071] = {X 354.8685, Y 61.7063, Z -4.6667, A 0.000, B 0.000, C 0.000 }
gfCNCPoint3[14072] = {X 352.3565, Y 62.1757, Z -4.6667, A 0.000, B 0.000, C 0.000 }
gfCNCPoint3[14073] = {X 349.8172, Y 62.4636, Z -4.6667, A 0.000, B 0.000, C 0.000 }
gfCNCPoint3[14074] = {X 347.2639, Y 62.5685, Z -4.6667, A 0.000, B 0.000, C 0.000 }
gfCNCPoint3[14075] = {X 345.1284, Y 62.5529, Z -4.6667, A 0.000, B 0.000, C 0.000 }
gfCNCPoint3[14076] = {X 342.9975, Y 62.4120, Z -4.6667, A 0.000, B 0.000, C 0.000 }
gfCNCPoint3[14077] = {X 340.8785, Y 62.1463, Z -4.6667, A 0.000, B 0.000, C 0.000 }
gfCNCPoint3[14078] = {X 340.4887, Y 63.7342, Z -4.6667, A 0.000, B 0.000, C 0.000 }
gfCNCPoint3[14079] = {X 339.9474, Y 65.2770, Z -4.6667, A 0.000, B 0.000, C 0.000 }
gfCNCPoint3[14080] = {X 339.2597, Y 66.7604, Z -4.6667, A 0.000, B 0.000, C 0.000 }
gfCNCPoint3[14081] = {X 338.4320, Y 68.1704, Z -4.6667, A 0.000, B 0.000, C 0.000 }
gfCNCPoint3[14082] = {X 337.4721, Y 69.4940, Z -4.6667, A 0.000, B 0.000, C 0.000 }
gfCNCPoint3[14083] = {X 337.4728, Y 77.4158, Z -4.6667, A 0.000, B 0.000, C 0.000 }
gfCNCPoint3[14084] = {X 340.9055, Y 77.6559, Z -4.6667, A 0.000, B 0.000, C 0.000 }
gfCNCPoint3[14085] = {X 344.3441, Y 77.7883, Z -4.6667, A 0.000, B 0.000, C 0.000 }
gfCNCPoint3[14086] = {X 347.7851, Y 77.8129, Z -4.6667, A 0.000, B 0.000, C 0.000 }
gfCNCPoint3[14087] = {X 351.3137, Y 77.7920, Z -4.6667, A 0.000, B 0.000, C 0.000 }
gfCNCPoint3[14088] = {X 354.8398, Y 77.6573, Z -4.6667, A 0.000, B 0.000, C 0.000 }
gfCNCPoint3[14089] = {X 358.3596, Y 77.4088, Z -4.6667, A 0.000, B 0.000, C 0.000 }
gfCNCPoint3[14090] = {X 358.3591, Y 69.5049, Z -4.6667, A 0.000, B 0.000, C 0.000 }
gfCNCPoint3[14091] = {X 357.3030, Y 68.0353, Z -4.6667, A 0.000, B 0.000, C 0.000 }
gfCNCPoint3[14092] = {X 356.4104, Y 66.4610, Z -4.6667, A 0.000, B 0.000, C 0.000 }
gfCNCPoint3[14093] = {X 358.5585, Y 65.3908, Z -4.6667, A 0.000, B 0.000, C 0.000 }
gfCNCPoint3[14094] = {X 357.9835, Y 64.0773, Z -4.6667, A 0.000, B 0.000, C 0.000 }
gfCNCPoint3[14095] = {X 357.5411, Y 62.7132, Z -4.6667, A 0.000, B 0.000, C 0.000 }
gfCNCPoint3[14096] = {X 357.2359, Y 61.3122, Z -4.6667, A 0.000, B 0.000, C 0.000 }
gfCNCPoint3[14097] = {X 357.0916, Y 60.1637, Z -4.6667, A 0.000, B 0.000, C 0.000 }
gfCNCPoint3[14098] = {X 357.0395, Y 59.0073, Z -4.6667, A 0.000, B 0.000, C 0.000 }
gfCNCPoint3[14099] = {X 357.0394, Y 58.6394, Z -4.6667, A 0.000, B 0.000, C 0.000 }
gfCNCPoint3[14100] = {X 355.6989, Y 59.0303, Z -4.6667, A 0.000, B 0.000, C 0.000 }
gfCNCPoint3[14101] = {X 354.3432, Y 59.3645, Z -4.6667, A 0.000, B 0.000, C 0.000 }
gfCNCPoint3[14102] = {X 351.9939, Y 59.8032, Z -4.6667, A 0.000, B 0.000, C 0.000 }
gfCNCPoint3[14103] = {X 349.6192, Y 60.0717, Z -4.6667, A 0.000, B 0.000, C 0.000 }
gfCNCPoint3[14104] = {X 347.2313, Y 60.1686, Z -4.6667, A 0.000, B 0.000, C 0.000 }
gfCNCPoint3[14105] = {X 344.3951, Y 60.1145, Z -4.6667, A 0.000, B 0.000, C 0.000 }
gfCNCPoint3[14106] = {X 341.5733, Y 59.8239, Z -4.6667, A 0.000, B 0.000, C 0.000 }
gfCNCPoint3[14107] = {X 338.7856, Y 59.2988, Z -4.6667, A 0.000, B 0.000, C 0.000 }
gfCNCPoint3[14108] = {X 338.6399, Y 60.9981, Z -4.6667, A 0.000, B 0.000, C 0.000 }
gfCNCPoint3[14109] = {X 338.2960, Y 62.6687, Z -4.6667, A 0.000, B 0.000, C 0.000 }
gfCNCPoint3[14110] = {X 337.7586, Y 64.2873, Z -4.6667, A 0.000, B 0.000, C 0.000 }
gfCNCPoint3[14111] = {X 337.0351, Y 65.8318, Z -4.6667, A 0.000, B 0.000, C 0.000 }
gfCNCPoint3[14112] = {X 336.1354, Y 67.2807, Z -4.6667, A 0.000, B 0.000, C 0.000 }
gfCNCPoint3[14113] = {X 335.0720, Y 68.6142, Z -4.6667, A 0.000, B 0.000, C 0.000 }
gfCNCPoint3[14114] = {X 335.0729, Y 79.5883, Z -4.6667, A 0.000, B 0.000, C 0.000 }
gfCNCPoint3[14115] = {X 335.6632, Y 79.6572, Z -4.6667, A 0.000, B 0.000, C 0.000 }
gfCNCPoint3[14116] = {X 336.2545, Y 79.7156, Z -4.6667, A 0.000, B 0.000, C 0.000 }
gfCNCPoint3[14117] = {X 340.0909, Y 80.0131, Z -4.6667, A 0.000, B 0.000, C 0.000 }
gfCNCPoint3[14118] = {X 343.9353, Y 80.1790, Z -4.6667, A 0.000, B 0.000, C 0.000 }
gfCNCPoint3[14119] = {X 347.7831, Y 80.2130, Z -4.6667, A 0.000, B 0.000, C 0.000 }
gfCNCPoint3[14120] = {X 351.8382, Y 80.1801, Z -4.6667, A 0.000, B 0.000, C 0.000 }
gfCNCPoint3[14121] = {X 355.8895, Y 80.0000, Z -4.6667, A 0.000, B 0.000, C 0.000 }
gfCNCPoint3[14122] = {X 359.9315, Y 79.6729, Z -4.6667, A 0.000, B 0.000, C 0.000 }
gfCNCPoint3[14123] = {X 360.3460, Y 79.6313, Z -4.6667, A 0.000, B 0.000, C 0.000 }
gfCNCPoint3[14124] = {X 360.7598, Y 79.5837, Z -4.6667, A 0.000, B 0.000, C 0.000 }
gfCNCPoint3[14125] = {X 360.7590, Y 68.6236, Z -4.6667, A 0.000, B 0.000, C 0.000 }
gfCNCPoint3[14126] = {X 359.9291, Y 67.6138, Z -4.6667, A 0.000, B 0.000, C 0.000 }
gfCNCPoint3[14127] = {X 359.1936, Y 66.5333, Z -4.6667, A 0.000, B 0.000, C 0.000 }
gfCNCPoint3[14128] = {X 358.5585, Y 65.3908, Z -4.6667, A 0.000, B 0.000, C 0.000 }
gfCNCPoint3[14129] = {X 360.7067, Y 64.3207, Z -4.6667, A 0.000, B 0.000, C 0.000 }
gfCNCPoint3[14130] = {X 360.1635, Y 63.0538, Z -4.6667, A 0.000, B 0.000, C 0.000 }
gfCNCPoint3[14131] = {X 359.7681, Y 61.7332, Z -4.6667, A 0.000, B 0.000, C 0.000 }
gfCNCPoint3[14132] = {X 359.5257, Y 60.3763, Z -4.6667, A 0.000, B 0.000, C 0.000 }
gfCNCPoint3[14133] = {X 359.4395, Y 59.0005, Z -4.6667, A 0.000, B 0.000, C 0.000 }
gfCNCPoint3[14134] = {X 359.4393, Y 58.0000, Z -4.6667, A 0.000, B 0.000, C 0.000 }
gfCNCPoint3[14135] = {X 359.5343, Y 56.4880, Z -4.6667, A 0.000, B 0.000, C 0.000 }
gfCNCPoint3[14136] = {X 359.8178, Y 54.9997, Z -4.6667, A 0.000, B 0.000, C 0.000 }
gfCNCPoint3[14137] = {X 359.3651, Y 55.2117, Z -4.6667, A 0.000, B 0.000, C 0.000 }
gfCNCPoint3[14138] = {X 357.8572, Y 55.8211, Z -4.6667, A 0.000, B 0.000, C 0.000 }
gfCNCPoint3[14139] = {X 356.3191, Y 56.3500, Z -4.6667, A 0.000, B 0.000, C 0.000 }
gfCNCPoint3[14140] = {X 354.0856, Y 56.9614, Z -4.6667, A 0.000, B 0.000, C 0.000 }
gfCNCPoint3[14141] = {X 351.8124, Y 57.4032, Z -4.6667, A 0.000, B 0.000, C 0.000 }
gfCNCPoint3[14142] = {X 349.5124, Y 57.6728, Z -4.6667, A 0.000, B 0.000, C 0.000 }
gfCNCPoint3[14143] = {X 347.1986, Y 57.7687, Z -4.6667, A 0.000, B 0.000, C 0.000 }
gfCNCPoint3[14144] = {X 344.5555, Y 57.7198, Z -4.6667, A 0.000, B 0.000, C 0.000 }
gfCNCPoint3[14145] = {X 341.9258, Y 57.4499, Z -4.6667, A 0.000, B 0.000, C 0.000 }
gfCNCPoint3[14146] = {X 339.3279, Y 56.9609, Z -4.6667, A 0.000, B 0.000, C 0.000 }
gfCNCPoint3[14147] = {X 337.7709, Y 56.5577, Z -4.6667, A 0.000, B 0.000, C 0.000 }
gfCNCPoint3[14148] = {X 336.2364, Y 56.0757, Z -4.6667, A 0.000, B 0.000, C 0.000 }
gfCNCPoint3[14149] = {X 336.3521, Y 57.0348, Z -4.6667, A 0.000, B 0.000, C 0.000 }
gfCNCPoint3[14150] = {X 336.3907, Y 58.0000, Z -4.6667, A 0.000, B 0.000, C 0.000 }
gfCNCPoint3[14151] = {X 336.3907, Y 58.9527, Z -4.6667, A 0.000, B 0.000, C 0.000 }
gfCNCPoint3[14152] = {X 336.3894, Y 59.0937, Z -4.6667, A 0.000, B 0.000, C 0.000 }
gfCNCPoint3[14153] = {X 336.3864, Y 59.2347, Z -4.6667, A 0.000, B 0.000, C 0.000 }
gfCNCPoint3[14154] = {X 336.2428, Y 60.7989, Z -4.6667, A 0.000, B 0.000, C 0.000 }
gfCNCPoint3[14155] = {X 335.8980, Y 62.3314, Z -4.6667, A 0.000, B 0.000, C 0.000 }
gfCNCPoint3[14156] = {X 335.3580, Y 63.8064, Z -4.6667, A 0.000, B 0.000, C 0.000 }
gfCNCPoint3[14157] = {X 334.6316, Y 65.1992, Z -4.6667, A 0.000, B 0.000, C 0.000 }
gfCNCPoint3[14158] = {X 333.7312, Y 66.4863, Z -4.6667, A 0.000, B 0.000, C 0.000 }
gfCNCPoint3[14159] = {X 332.6719, Y 67.6462, Z -4.6667, A 0.000, B 0.000, C 0.000 }
gfCNCPoint3[14160] = {X 332.6731, Y 81.6417, Z -4.6667, A 0.000, B 0.000, C 0.000 }
gfCNCPoint3[14161] = {X 334.3509, Y 81.9138, Z -4.6667, A 0.000, B 0.000, C 0.000 }
gfCNCPoint3[14162] = {X 336.0397, Y 82.1060, Z -4.6667, A 0.000, B 0.000, C 0.000 }
gfCNCPoint3[14163] = {X 339.9469, Y 82.4088, Z -4.6667, A 0.000, B 0.000, C 0.000 }
gfCNCPoint3[14164] = {X 343.8622, Y 82.5779, Z -4.6667, A 0.000, B 0.000, C 0.000 }
gfCNCPoint3[14165] = {X 347.7810, Y 82.6131, Z -4.6667, A 0.000, B 0.000, C 0.000 }
gfCNCPoint3[14166] = {X 351.9135, Y 82.5789, Z -4.6667, A 0.000, B 0.000, C 0.000 }
gfCNCPoint3[14167] = {X 356.0421, Y 82.3951, Z -4.6667, A 0.000, B 0.000, C 0.000 }
gfCNCPoint3[14168] = {X 360.1614, Y 82.0619, Z -4.6667, A 0.000, B 0.000, C 0.000 }
gfCNCPoint3[14169] = {X 361.6659, Y 81.8844, Z -4.6667, A 0.000, B 0.000, C 0.000 }
gfCNCPoint3[14170] = {X 363.1599, Y 81.6337, Z -4.6667, A 0.000, B 0.000, C 0.000 }
gfCNCPoint3[14171] = {X 363.1589, Y 67.6537, Z -4.6667, A 0.000, B 0.000, C 0.000 }
gfCNCPoint3[14172] = {X 362.2156, Y 66.6391, Z -4.6667, A 0.000, B 0.000, C 0.000 }
gfCNCPoint3[14173] = {X 361.3946, Y 65.5232, Z -4.6667, A 0.000, B 0.000, C 0.000 }
gfCNCPoint3[14174] = {X 360.7067, Y 64.3207, Z -4.6667, A 0.000, B 0.000, C 0.000 }
gfCNCPoint3[14175] = {X 362.8549, Y 63.2505, Z -4.6667, A 0.000, B 0.000, C 0.000 }
gfCNCPoint3[14176] = {X 362.3011, Y 61.8885, Z -4.6667, A 0.000, B 0.000, C 0.000 }
gfCNCPoint3[14177] = {X 361.9600, Y 60.4583, Z -4.6667, A 0.000, B 0.000, C 0.000 }
gfCNCPoint3[14178] = {X 361.8395, Y 58.9930, Z -4.6667, A 0.000, B 0.000, C 0.000 }
gfCNCPoint3[14179] = {X 361.8393, Y 58.0000, Z -4.6667, A 0.000, B 0.000, C 0.000 }
gfCNCPoint3[14180] = {X 361.9154, Y 56.7884, Z -4.6667, A 0.000, B 0.000, C 0.000 }
gfCNCPoint3[14181] = {X 362.1426, Y 55.5958, Z -4.6667, A 0.000, B 0.000, C 0.000 }
gfCNCPoint3[14182] = {X 362.5739, Y 54.3010, Z -4.6667, A 0.000, B 0.000, C 0.000 }
gfCNCPoint3[14183] = {X 363.1830, Y 53.0797, Z -4.6667, A 0.000, B 0.000, C 0.000 }
gfCNCPoint3[14184] = {X 363.9578, Y 51.9562, Z -4.6667, A 0.000, B 0.000, C 0.000 }
gfCNCPoint3[14185] = {X 364.8830, Y 50.9529, Z -4.6667, A 0.000, B 0.000, C 0.000 }
gfCNCPoint3[14186] = {X 365.9400, Y 50.0896, Z -4.6667, A 0.000, B 0.000, C 0.000 }
gfCNCPoint3[14187] = {X 367.1079, Y 49.3836, Z -4.6667, A 0.000, B 0.000, C 0.000 }
gfCNCPoint3[14188] = {X 368.3636, Y 48.8488, Z -4.6667, A 0.000, B 0.000, C 0.000 }
gfCNCPoint3[14189] = {X 369.6819, Y 48.4960, Z -4.6667, A 0.000, B 0.000, C 0.000 }
gfCNCPoint3[14190] = {X 371.0368, Y 48.3320, Z -4.6667, A 0.000, B 0.000, C 0.000 }
gfCNCPoint3[14191] = {X 371.2780, Y 48.3230, Z -4.6667, A 0.000, B 0.000, C 0.000 }
gfCNCPoint3[14192] = {X 371.5193, Y 48.3200, Z -4.6667, A 0.000, B 0.000, C 0.000 }
gfCNCPoint3[14193] = {X 388.0597, Y 48.3200, Z -4.6667, A 0.000, B 0.000, C 0.000 }
gfCNCPoint3[14194] = {X 389.4419, Y 48.4192, Z -4.6667, A 0.000, B 0.000, C 0.000 }
gfCNCPoint3[14195] = {X 390.7958, Y 48.7147, Z -4.6667, A 0.000, B 0.000, C 0.000 }
gfCNCPoint3[14196] = {X 392.0936, Y 49.2006, Z -4.6667, A 0.000, B 0.000, C 0.000 }
gfCNCPoint3[14197] = {X 393.3087, Y 49.8667, Z -4.6667, A 0.000, B 0.000, C 0.000 }
gfCNCPoint3[14198] = {X 394.5333, Y 49.1962, Z -4.6667, A 0.000, B 0.000, C 0.000 }
gfCNCPoint3[14199] = {X 395.8416, Y 48.7089, Z -4.6667, A 0.000, B 0.000, C 0.000 }
gfCNCPoint3[14200] = {X 397.1858, Y 48.4177, Z -4.6667, A 0.000, B 0.000, C 0.000 }
gfCNCPoint3[14201] = {X 398.5577, Y 48.3200, Z -4.6667, A 0.000, B 0.000, C 0.000 }
gfCNCPoint3[14202] = {X 398.7346, Y 48.3200, Z -4.6667, A 0.000, B 0.000, C 0.000 }
gfCNCPoint3[14203] = {X 398.1859, Y 47.6069, Z -4.6667, A 0.000, B 0.000, C 0.000 }
gfCNCPoint3[14204] = {X 397.7774, Y 46.8051, Z -4.6667, A 0.000, B 0.000, C 0.000 }
gfCNCPoint3[14205] = {X 397.5230, Y 45.9420, Z -4.6667, A 0.000, B 0.000, C 0.000 }
gfCNCPoint3[14206] = {X 397.4561, Y 45.4921, Z -4.6667, A 0.000, B 0.000, C 0.000 }
gfCNCPoint3[14207] = {X 397.4314, Y 45.0378, Z -4.6667, A 0.000, B 0.000, C 0.000 }
gfCNCPoint3[14208] = {X 397.4316, Y 44.1456, Z -4.6667, A 0.000, B 0.000, C 0.000 }
gfCNCPoint3[14209] = {X 397.5413, Y 43.1780, Z -4.6667, A 0.000, B 0.000, C 0.000 }
gfCNCPoint3[14210] = {X 397.8410, Y 42.2514, Z -4.6667, A 0.000, B 0.000, C 0.000 }
gfCNCPoint3[14211] = {X 398.3186, Y 41.4029, Z -4.6667, A 0.000, B 0.000, C 0.000 }
gfCNCPoint3[14212] = {X 398.9552, Y 40.6660, Z -4.6667, A 0.000, B 0.000, C 0.000 }
gfCNCPoint3[14213] = {X 398.9552, Y 31.8235, Z -4.6667, A 0.000, B 0.000, C 0.000 }
gfCNCPoint3[14214] = {X 396.7502, Y 27.9891, Z -4.6667, A 0.000, B 0.000, C 0.000 }
gfCNCPoint3[14215] = {X 386.3476, Y 33.9712, Z -4.6667, A 0.000, B 0.000, C 0.000 }
gfCNCPoint3[14216] = {X 386.2667, Y 34.3983, Z -4.6667, A 0.000, B 0.000, C 0.000 }
gfCNCPoint3[14217] = {X 386.1821, Y 34.8245, Z -4.6667, A 0.000, B 0.000, C 0.000 }
gfCNCPoint3[14218] = {X 386.0230, Y 35.5738, Z -4.6667, A 0.000, B 0.000, C 0.000 }
gfCNCPoint3[14219] = {X 385.8503, Y 36.3200, Z -4.6667, A 0.000, B 0.000, C 0.000 }
gfCNCPoint3[14220] = {X 386.9552, Y 36.3200, Z -4.6667, A 0.000, B 0.000, C 0.000 }
gfCNCPoint3[14221] = {X 386.9552, Y 35.0278, Z -4.6667, A 0.000, B 0.000, C 0.000 }
gfCNCPoint3[14222] = {X 386.3476, Y 33.9712, Z -4.6667, A 0.000, B 0.000, C 0.000 }
gfCNCPoint3[14223] = {X 388.4281, Y 32.7748, Z -4.6667, A 0.000, B 0.000, C 0.000 }
gfCNCPoint3[14224] = {X 384.7450, Y 26.3700, Z -4.6667, A 0.000, B 0.000, C 0.000 }
gfCNCPoint3[14225] = {X 384.6160, Y 28.7704, Z -4.6667, A 0.000, B 0.000, C 0.000 }
gfCNCPoint3[14226] = {X 384.3633, Y 31.1608, Z -4.6667, A 0.000, B 0.000, C 0.000 }
gfCNCPoint3[14227] = {X 383.9876, Y 33.5351, Z -4.6667, A 0.000, B 0.000, C 0.000 }
gfCNCPoint3[14228] = {X 383.9106, Y 33.9415, Z -4.6667, A 0.000, B 0.000, C 0.000 }
gfCNCPoint3[14229] = {X 383.8300, Y 34.3472, Z -4.6667, A 0.000, B 0.000, C 0.000 }
gfCNCPoint3[14230] = {X 383.6800, Y 35.0538, Z -4.6667, A 0.000, B 0.000, C 0.000 }
gfCNCPoint3[14231] = {X 383.5172, Y 35.7575, Z -4.6667, A 0.000, B 0.000, C 0.000 }
gfCNCPoint3[14232] = {X 383.1272, Y 37.2469, Z -4.6667, A 0.000, B 0.000, C 0.000 }
gfCNCPoint3[14233] = {X 382.6795, Y 38.7200, Z -4.6667, A 0.000, B 0.000, C 0.000 }
gfCNCPoint3[14234] = {X 388.0597, Y 38.7200, Z -4.6667, A 0.000, B 0.000, C 0.000 }
gfCNCPoint3[14235] = {X 388.4821, Y 38.7246, Z -4.6667, A 0.000, B 0.000, C 0.000 }
gfCNCPoint3[14236] = {X 388.9043, Y 38.7385, Z -4.6667, A 0.000, B 0.000, C 0.000 }
gfCNCPoint3[14237] = {X 389.1204, Y 38.2363, Z -4.6667, A 0.000, B 0.000, C 0.000 }
gfCNCPoint3[14238] = {X 389.3552, Y 37.7427, Z -4.6667, A 0.000, B 0.000, C 0.000 }
gfCNCPoint3[14239] = {X 389.3552, Y 34.3869, Z -4.6667, A 0.000, B 0.000, C 0.000 }
gfCNCPoint3[14240] = {X 388.4281, Y 32.7748, Z -4.6667, A 0.000, B 0.000, C 0.000 }
gfCNCPoint3[14241] = {X 390.5086, Y 31.5784, Z -4.6667, A 0.000, B 0.000, C 0.000 }
gfCNCPoint3[14242] = {X 386.7884, Y 25.1090, Z -4.6667, A 0.000, B 0.000, C 0.000 }
gfCNCPoint3[14243] = {X 386.1511, Y 24.0198, Z -4.6667, A 0.000, B 0.000, C 0.000 }
gfCNCPoint3[14244] = {X 385.4975, Y 22.9404, Z -4.6667, A 0.000, B 0.000, C 0.000 }
gfCNCPoint3[14245] = {X 384.4694, Y 22.1510, Z -4.6667, A 0.000, B 0.000, C 0.000 }
gfCNCPoint3[14246] = {X 383.5317, Y 21.2559, Z -4.6667, A 0.000, B 0.000, C 0.000 }
gfCNCPoint3[14247] = {X 382.6954, Y 20.2655, Z -4.6667, A 0.000, B 0.000, C 0.000 }
gfCNCPoint3[14248] = {X 381.9700, Y 19.1913, Z -4.6667, A 0.000, B 0.000, C 0.000 }
gfCNCPoint3[14249] = {X 382.2229, Y 21.5540, Z -4.6667, A 0.000, B 0.000, C 0.000 }
gfCNCPoint3[14250] = {X 382.3483, Y 23.9269, Z -4.6667, A 0.000, B 0.000, C 0.000 }
gfCNCPoint3[14251] = {X 382.3459, Y 26.3031, Z -4.6667, A 0.000, B 0.000, C 0.000 }
gfCNCPoint3[14252] = {X 382.2020, Y 28.8406, Z -4.6667, A 0.000, B 0.000, C 0.000 }
gfCNCPoint3[14253] = {X 381.9124, Y 31.3656, Z -4.6667, A 0.000, B 0.000, C 0.000 }
gfCNCPoint3[14254] = {X 381.4780, Y 33.8698, Z -4.6667, A 0.000, B 0.000, C 0.000 }
gfCNCPoint3[14255] = {X 380.9965, Y 35.9391, Z -4.6667, A 0.000, B 0.000, C 0.000 }
gfCNCPoint3[14256] = {X 380.3973, Y 37.9775, Z -4.6667, A 0.000, B 0.000, C 0.000 }
gfCNCPoint3[14257] = {X 379.8417, Y 39.5621, Z -4.6667, A 0.000, B 0.000, C 0.000 }
gfCNCPoint3[14258] = {X 379.2150, Y 41.1200, Z -4.6667, A 0.000, B 0.000, C 0.000 }
gfCNCPoint3[14259] = {X 388.0597, Y 41.1200, Z -4.6667, A 0.000, B 0.000, C 0.000 }
gfCNCPoint3[14260] = {X 389.3256, Y 41.1675, Z -4.6667, A 0.000, B 0.000, C 0.000 }
gfCNCPoint3[14261] = {X 390.5843, Y 41.3099, Z -4.6667, A 0.000, B 0.000, C 0.000 }
gfCNCPoint3[14262] = {X 391.0709, Y 39.7838, Z -4.6667, A 0.000, B 0.000, C 0.000 }
gfCNCPoint3[14263] = {X 391.7552, Y 38.3355, Z -4.6667, A 0.000, B 0.000, C 0.000 }
gfCNCPoint3[14264] = {X 391.7552, Y 33.7461, Z -4.6667, A 0.000, B 0.000, C 0.000 }
gfCNCPoint3[14265] = {X 390.5086, Y 31.5784, Z -4.6667, A 0.000, B 0.000, C 0.000 }
gfCNCPoint3[14266] = {X 392.5892, Y 30.3820, Z -4.6667, A 0.000, B 0.000, C 0.000 }
gfCNCPoint3[14267] = {X 388.8689, Y 23.9126, Z -4.6667, A 0.000, B 0.000, C 0.000 }
gfCNCPoint3[14268] = {X 388.0745, Y 22.5598, Z -4.6667, A 0.000, B 0.000, C 0.000 }
gfCNCPoint3[14269] = {X 387.2557, Y 21.2217, Z -4.6667, A 0.000, B 0.000, C 0.000 }
gfCNCPoint3[14270] = {X 386.3076, Y 20.5567, Z -4.6667, A 0.000, B 0.000, C 0.000 }
gfCNCPoint3[14271] = {X 385.4456, Y 19.7834, Z -4.6667, A 0.000, B 0.000, C 0.000 }
gfCNCPoint3[14272] = {X 384.6822, Y 18.9126, Z -4.6667, A 0.000, B 0.000, C 0.000 }
gfCNCPoint3[14273] = {X 384.0282, Y 17.9568, Z -4.6667, A 0.000, B 0.000, C 0.000 }
gfCNCPoint3[14274] = {X 383.4399, Y 16.8089, Z -4.6667, A 0.000, B 0.000, C 0.000 }
gfCNCPoint3[14275] = {X 383.0095, Y 15.5930, Z -4.6667, A 0.000, B 0.000, C 0.000 }
gfCNCPoint3[14276] = {X 382.7446, Y 14.3307, Z -4.6667, A 0.000, B 0.000, C 0.000 }
gfCNCPoint3[14277] = {X 382.6498, Y 13.0443, Z -4.6667, A 0.000, B 0.000, C 0.000 }
gfCNCPoint3[14278] = {X 382.6496, Y 12.1868, Z -4.6667, A 0.000, B 0.000, C 0.000 }
gfCNCPoint3[14279] = {X 382.6507, Y 12.0459, Z -4.6667, A 0.000, B 0.000, C 0.000 }
gfCNCPoint3[14280] = {X 382.6537, Y 11.9050, Z -4.6667, A 0.000, B 0.000, C 0.000 }
gfCNCPoint3[14281] = {X 377.7927, Y 11.9050, Z -4.6667, A 0.000, B 0.000, C 0.000 }
gfCNCPoint3[14282] = {X 378.4141, Y 13.8379, Z -4.6667, A 0.000, B 0.000, C 0.000 }
gfCNCPoint3[14283] = {X 378.9221, Y 15.8037, Z -4.6667, A 0.000, B 0.000, C 0.000 }
gfCNCPoint3[14284] = {X 379.2985, Y 17.6497, Z -4.6667, A 0.000, B 0.000, C 0.000 }
gfCNCPoint3[14285] = {X 379.5913, Y 19.5108, Z -4.6667, A 0.000, B 0.000, C 0.000 }
gfCNCPoint3[14286] = {X 379.8702, Y 22.2871, Z -4.6667, A 0.000, B 0.000, C 0.000 }
gfCNCPoint3[14287] = {X 379.9631, Y 25.0759, Z -4.6667, A 0.000, B 0.000, C 0.000 }
gfCNCPoint3[14288] = {X 379.8696, Y 27.8646, Z -4.6667, A 0.000, B 0.000, C 0.000 }
gfCNCPoint3[14289] = {X 379.5901, Y 30.6409, Z -4.6667, A 0.000, B 0.000, C 0.000 }
gfCNCPoint3[14290] = {X 379.1259, Y 33.3924, Z -4.6667, A 0.000, B 0.000, C 0.000 }
gfCNCPoint3[14291] = {X 378.5757, Y 35.6995, Z -4.6667, A 0.000, B 0.000, C 0.000 }
gfCNCPoint3[14292] = {X 377.8690, Y 37.9636, Z -4.6667, A 0.000, B 0.000, C 0.000 }
gfCNCPoint3[14293] = {X 377.0093, Y 40.1741, Z -4.6667, A 0.000, B 0.000, C 0.000 }
gfCNCPoint3[14294] = {X 376.2276, Y 41.8693, Z -4.6667, A 0.000, B 0.000, C 0.000 }
gfCNCPoint3[14295] = {X 375.3559, Y 43.5200, Z -4.6667, A 0.000, B 0.000, C 0.000 }
gfCNCPoint3[14296] = {X 388.0597, Y 43.5200, Z -4.6667, A 0.000, B 0.000, C 0.000 }
gfCNCPoint3[14297] = {X 389.6072, Y 43.6029, Z -4.6667, A 0.000, B 0.000, C 0.000 }
gfCNCPoint3[14298] = {X 391.1370, Y 43.8508, Z -4.6667, A 0.000, B 0.000, C 0.000 }
gfCNCPoint3[14299] = {X 392.6316, Y 44.2607, Z -4.6667, A 0.000, B 0.000, C 0.000 }
gfCNCPoint3[14300] = {X 392.7236, Y 42.8756, Z -4.6667, A 0.000, B 0.000, C 0.000 }
gfCNCPoint3[14301] = {X 393.0129, Y 41.5179, Z -4.6667, A 0.000, B 0.000, C 0.000 }
gfCNCPoint3[14302] = {X 393.4934, Y 40.2155, Z -4.6667, A 0.000, B 0.000, C 0.000 }
gfCNCPoint3[14303] = {X 394.1552, Y 38.9952, Z -4.6667, A 0.000, B 0.000, C 0.000 }
gfCNCPoint3[14304] = {X 394.1552, Y 33.1052, Z -4.6667, A 0.000, B 0.000, C 0.000 }
gfCNCPoint3[14305] = {X 392.5892, Y 30.3820, Z -4.6667, A 0.000, B 0.000, C 0.000 }
gfCNCPoint3[14306] = {X 394.6697, Y 29.1855, Z -4.6667, A 0.000, B 0.000, C 0.000 }
gfCNCPoint3[14307] = {X 390.9494, Y 22.7161, Z -4.6667, A 0.000, B 0.000, C 0.000 }
gfCNCPoint3[14308] = {X 390.0906, Y 21.2552, Z -4.6667, A 0.000, B 0.000, C 0.000 }
gfCNCPoint3[14309] = {X 389.2040, Y 19.8109, Z -4.6667, A 0.000, B 0.000, C 0.000 }
gfCNCPoint3[14310] = {X 389.0618, Y 19.6012, Z -4.6667, A 0.000, B 0.000, C 0.000 }
gfCNCPoint3[14311] = {X 388.9049, Y 19.4022, Z -4.6667, A 0.000, B 0.000, C 0.000 }
gfCNCPoint3[14312] = {X 387.8166, Y 18.6904, Z -4.6667, A 0.000, B 0.000, C 0.000 }
gfCNCPoint3[14313] = {X 386.8722, Y 17.7962, Z -4.6667, A 0.000, B 0.000, C 0.000 }
gfCNCPoint3[14314] = {X 386.1020, Y 16.7484, Z -4.6667, A 0.000, B 0.000, C 0.000 }
gfCNCPoint3[14315] = {X 385.5306, Y 15.5802, Z -4.6667, A 0.000, B 0.000, C 0.000 }
gfCNCPoint3[14316] = {X 385.1761, Y 14.3290, Z -4.6667, A 0.000, B 0.000, C 0.000 }
gfCNCPoint3[14317] = {X 385.0498, Y 13.0347, Z -4.6667, A 0.000, B 0.000, C 0.000 }
gfCNCPoint3[14318] = {X 385.0496, Y 12.1868, Z -4.6667, A 0.000, B 0.000, C 0.000 }
gfCNCPoint3[14319] = {X 385.0504, Y 12.0808, Z -4.6667, A 0.000, B 0.000, C 0.000 }
gfCNCPoint3[14320] = {X 385.0527, Y 11.9749, Z -4.6667, A 0.000, B 0.000, C 0.000 }
gfCNCPoint3[14321] = {X 385.1994, Y 10.7177, Z -4.6667, A 0.000, B 0.000, C 0.000 }
gfCNCPoint3[14322] = {X 385.5616, Y 9.5050, Z -4.6667, A 0.000, B 0.000, C 0.000 }
gfCNCPoint3[14323] = {X 374.2012, Y 9.5050, Z -4.6667, A 0.000, B 0.000, C 0.000 }
gfCNCPoint3[14324] = {X 374.9084, Y 11.0876, Z -4.6667, A 0.000, B 0.000, C 0.000 }
gfCNCPoint3[14325] = {X 375.5302, Y 12.7057, Z -4.6667, A 0.000, B 0.000, C 0.000 }
gfCNCPoint3[14326] = {X 376.1089, Y 14.5057, Z -4.6667, A 0.000, B 0.000, C 0.000 }
gfCNCPoint3[14327] = {X 376.5819, Y 16.3362, Z -4.6667, A 0.000, B 0.000, C 0.000 }
gfCNCPoint3[14328] = {X 377.1031, Y 19.0706, Z -4.6667, A 0.000, B 0.000, C 0.000 }
gfCNCPoint3[14329] = {X 377.4299, Y 21.8349, Z -4.6667, A 0.000, B 0.000, C 0.000 }
gfCNCPoint3[14330] = {X 377.5605, Y 24.6154, Z -4.6667, A 0.000, B 0.000, C 0.000 }
gfCNCPoint3[14331] = {X 377.4943, Y 27.3981, Z -4.6667, A 0.000, B 0.000, C 0.000 }
gfCNCPoint3[14332] = {X 377.2317, Y 30.1693, Z -4.6667, A 0.000, B 0.000, C 0.000 }
gfCNCPoint3[14333] = {X 376.7739, Y 32.9150, Z -4.6667, A 0.000, B 0.000, C 0.000 }
gfCNCPoint3[14334] = {X 376.1762, Y 35.3677, Z -4.6667, A 0.000, B 0.000, C 0.000 }
gfCNCPoint3[14335] = {X 375.3887, Y 37.7663, Z -4.6667, A 0.000, B 0.000, C 0.000 }
gfCNCPoint3[14336] = {X 374.4162, Y 40.0960, Z -4.6667, A 0.000, B 0.000, C 0.000 }
gfCNCPoint3[14337] = {X 373.2646, Y 42.3426, Z -4.6667, A 0.000, B 0.000, C 0.000 }
gfCNCPoint3[14338] = {X 372.1960, Y 44.1063, Z -4.6667, A 0.000, B 0.000, C 0.000 }
gfCNCPoint3[14339] = {X 371.0170, Y 45.7982, Z -4.6667, A 0.000, B 0.000, C 0.000 }
gfCNCPoint3[14340] = {X 370.9172, Y 45.9350, Z -4.6667, A 0.000, B 0.000, C 0.000 }
gfCNCPoint3[14341] = {X 371.2181, Y 45.9238, Z -4.6667, A 0.000, B 0.000, C 0.000 }
gfCNCPoint3[14342] = {X 371.5193, Y 45.9200, Z -4.6667, A 0.000, B 0.000, C 0.000 }
gfCNCPoint3[14343] = {X 388.0597, Y 45.9200, Z -4.6667, A 0.000, B 0.000, C 0.000 }
gfCNCPoint3[14344] = {X 389.4143, Y 45.9962, Z -4.6667, A 0.000, B 0.000, C 0.000 }
gfCNCPoint3[14345] = {X 390.7519, Y 46.2238, Z -4.6667, A 0.000, B 0.000, C 0.000 }
gfCNCPoint3[14346] = {X 392.0555, Y 46.6000, Z -4.6667, A 0.000, B 0.000, C 0.000 }
gfCNCPoint3[14347] = {X 393.3087, Y 47.1200, Z -4.6667, A 0.000, B 0.000, C 0.000 }
gfCNCPoint3[14348] = {X 394.2237, Y 46.7243, Z -4.6667, A 0.000, B 0.000, C 0.000 }
gfCNCPoint3[14349] = {X 395.1681, Y 46.4053, Z -4.6667, A 0.000, B 0.000, C 0.000 }
gfCNCPoint3[14350] = {X 395.0678, Y 45.7292, Z -4.6667, A 0.000, B 0.000, C 0.000 }
gfCNCPoint3[14351] = {X 395.0314, Y 45.0468, Z -4.6667, A 0.000, B 0.000, C 0.000 }
gfCNCPoint3[14352] = {X 395.0316, Y 44.1297, Z -4.6667, A 0.000, B 0.000, C 0.000 }
gfCNCPoint3[14353] = {X 395.1397, Y 42.9565, Z -4.6667, A 0.000, B 0.000, C 0.000 }
gfCNCPoint3[14354] = {X 395.4356, Y 41.8161, Z -4.6667, A 0.000, B 0.000, C 0.000 }
gfCNCPoint3[14355] = {X 395.9116, Y 40.7384, Z -4.6667, A 0.000, B 0.000, C 0.000 }
gfCNCPoint3[14356] = {X 396.5552, Y 39.7516, Z -4.6667, A 0.000, B 0.000, C 0.000 }
gfCNCPoint3[14357] = {X 396.5552, Y 32.4643, Z -4.6667, A 0.000, B 0.000, C 0.000 }
gfCNCPoint3[14358] = {X 394.6697, Y 29.1855, Z -4.6667, A 0.000, B 0.000, C 0.000 }
gfCNCPoint3[14359] = {X 396.7502, Y 27.9891, Z -4.6667, A 0.000, B 0.000, C 0.000 }
gfCNCPoint3[14360] = {X 393.0299, Y 21.5197, Z -4.6667, A 0.000, B 0.000, C 0.000 }
gfCNCPoint3[14361] = {X 392.1479, Y 20.0192, Z -4.6667, A 0.000, B 0.000, C 0.000 }
gfCNCPoint3[14362] = {X 391.2374, Y 18.5359, Z -4.6667, A 0.000, B 0.000, C 0.000 }
gfCNCPoint3[14363] = {X 390.8276, Y 17.9614, Z -4.6667, A 0.000, B 0.000, C 0.000 }
gfCNCPoint3[14364] = {X 390.3525, Y 17.4396, Z -4.6667, A 0.000, B 0.000, C 0.000 }
gfCNCPoint3[14365] = {X 389.5426, Y 16.9838, Z -4.6667, A 0.000, B 0.000, C 0.000 }
gfCNCPoint3[14366] = {X 388.8337, Y 16.3828, Z -4.6667, A 0.000, B 0.000, C 0.000 }
gfCNCPoint3[14367] = {X 388.2516, Y 15.6583, Z -4.6667, A 0.000, B 0.000, C 0.000 }
gfCNCPoint3[14368] = {X 387.8174, Y 14.8366, Z -4.6667, A 0.000, B 0.000, C 0.000 }
gfCNCPoint3[14369] = {X 387.5469, Y 13.9475, Z -4.6667, A 0.000, B 0.000, C 0.000 }
gfCNCPoint3[14370] = {X 387.4498, Y 13.0232, Z -4.6667, A 0.000, B 0.000, C 0.000 }
gfCNCPoint3[14371] = {X 387.4496, Y 12.1868, Z -4.6667, A 0.000, B 0.000, C 0.000 }
gfCNCPoint3[14372] = {X 387.5362, Y 11.2717, Z -4.6667, A 0.000, B 0.000, C 0.000 }
gfCNCPoint3[14373] = {X 387.7928, Y 10.3891, Z -4.6667, A 0.000, B 0.000, C 0.000 }
gfCNCPoint3[14374] = {X 388.2375, Y 9.5280, Z -4.6667, A 0.000, B 0.000, C 0.000 }
gfCNCPoint3[14375] = {X 388.8436, Y 8.7718, Z -4.6667, A 0.000, B 0.000, C 0.000 }
gfCNCPoint3[14376] = {X 389.5872, Y 8.1503, Z -4.6667, A 0.000, B 0.000, C 0.000 }
gfCNCPoint3[14377] = {X 390.4390, Y 7.6879, Z -4.6667, A 0.000, B 0.000, C 0.000 }
gfCNCPoint3[14378] = {X 391.3653, Y 7.4030, Z -4.6667, A 0.000, B 0.000, C 0.000 }
gfCNCPoint3[14379] = {X 392.3296, Y 7.3068, Z -4.6667, A 0.000, B 0.000, C 0.000 }
gfCNCPoint3[14380] = {X 399.1118, Y 7.3068, Z -4.6667, A 0.000, B 0.000, C 0.000 }
gfCNCPoint3[14381] = {X 400.0638, Y 7.4006, Z -4.6667, A 0.000, B 0.000, C 0.000 }
gfCNCPoint3[14382] = {X 400.9793, Y 7.6783, Z -4.6667, A 0.000, B 0.000, C 0.000 }
gfCNCPoint3[14383] = {X 401.8229, Y 8.1292, Z -4.6667, A 0.000, B 0.000, C 0.000 }
gfCNCPoint3[14384] = {X 402.5624, Y 8.7361, Z -4.6667, A 0.000, B 0.000, C 0.000 }
gfCNCPoint3[14385] = {X 403.1693, Y 9.4756, Z -4.6667, A 0.000, B 0.000, C 0.000 }
gfCNCPoint3[14386] = {X 403.6203, Y 10.3193, Z -4.6667, A 0.000, B 0.000, C 0.000 }
gfCNCPoint3[14387] = {X 403.8980, Y 11.2348, Z -4.6667, A 0.000, B 0.000, C 0.000 }
gfCNCPoint3[14388] = {X 403.9918, Y 12.1868, Z -4.6667, A 0.000, B 0.000, C 0.000 }
gfCNCPoint3[14389] = {X 403.9915, Y 13.0237, Z -4.6667, A 0.000, B 0.000, C 0.000 }
gfCNCPoint3[14390] = {X 403.9016, Y 13.9115, Z -4.6667, A 0.000, B 0.000, C 0.000 }
gfCNCPoint3[14391] = {X 403.6516, Y 14.7680, Z -4.6667, A 0.000, B 0.000, C 0.000 }
gfCNCPoint3[14392] = {X 405.3648, Y 17.7427, Z -4.6667, A 0.000, B 0.000, C 0.000 }
gfCNCPoint3[14393] = {X 407.2446, Y 14.6978, Z -4.6667, A 0.000, B 0.000, C 0.000 }
gfCNCPoint3[14394] = {X 407.0142, Y 13.8727, Z -4.6667, A 0.000, B 0.000, C 0.000 }
gfCNCPoint3[14395] = {X 406.9317, Y 13.0199, Z -4.6667, A 0.000, B 0.000, C 0.000 }
gfCNCPoint3[14396] = {X 406.9315, Y 12.1868, Z -4.6667, A 0.000, B 0.000, C 0.000 }
gfCNCPoint3[14397] = {X 407.0253, Y 11.2348, Z -4.6667, A 0.000, B 0.000, C 0.000 }
gfCNCPoint3[14398] = {X 407.3030, Y 10.3193, Z -4.6667, A 0.000, B 0.000, C 0.000 }
gfCNCPoint3[14399] = {X 407.7540, Y 9.4756, Z -4.6667, A 0.000, B 0.000, C 0.000 }
gfCNCPoint3[14400] = {X 408.3609, Y 8.7361, Z -4.6667, A 0.000, B 0.000, C 0.000 }
gfCNCPoint3[14401] = {X 409.1004, Y 8.1292, Z -4.6667, A 0.000, B 0.000, C 0.000 }
gfCNCPoint3[14402] = {X 409.9440, Y 7.6783, Z -4.6667, A 0.000, B 0.000, C 0.000 }
gfCNCPoint3[14403] = {X 410.8595, Y 7.4006, Z -4.6667, A 0.000, B 0.000, C 0.000 }
gfCNCPoint3[14404] = {X 411.8115, Y 7.3068, Z -4.6667, A 0.000, B 0.000, C 0.000 }
gfCNCPoint3[14405] = {X 419.3245, Y 7.3068, Z -4.6667, A 0.000, B 0.000, C 0.000 }
gfCNCPoint3[14406] = {X 420.2888, Y 7.4030, Z -4.6667, A 0.000, B 0.000, C 0.000 }
gfCNCPoint3[14407] = {X 421.2151, Y 7.6879, Z -4.6667, A 0.000, B 0.000, C 0.000 }
gfCNCPoint3[14408] = {X 422.0669, Y 8.1503, Z -4.6667, A 0.000, B 0.000, C 0.000 }
gfCNCPoint3[14409] = {X 422.8104, Y 8.7718, Z -4.6667, A 0.000, B 0.000, C 0.000 }
gfCNCPoint3[14410] = {X 423.4166, Y 9.5280, Z -4.6667, A 0.000, B 0.000, C 0.000 }
gfCNCPoint3[14411] = {X 423.8613, Y 10.3891, Z -4.6667, A 0.000, B 0.000, C 0.000 }
gfCNCPoint3[14412] = {X 424.1179, Y 11.2717, Z -4.6667, A 0.000, B 0.000, C 0.000 }
gfCNCPoint3[14413] = {X 424.2045, Y 12.1868, Z -4.6667, A 0.000, B 0.000, C 0.000 }
gfCNCPoint3[14414] = {X 424.2045, Y 12.9780, Z -4.6667, A 0.000, B 0.000, C 0.000 }
gfCNCPoint3[14415] = {X 424.1060, Y 13.9307, Z -4.6667, A 0.000, B 0.000, C 0.000 }
gfCNCPoint3[14416] = {X 423.8256, Y 14.8467, Z -4.6667, A 0.000, B 0.000, C 0.000 }
gfCNCPoint3[14417] = {X 423.3739, Y 15.6913, Z -4.6667, A 0.000, B 0.000, C 0.000 }
gfCNCPoint3[14418] = {X 422.7677, Y 16.4330, Z -4.6667, A 0.000, B 0.000, C 0.000 }
gfCNCPoint3[14419] = {X 422.0300, Y 17.0439, Z -4.6667, A 0.000, B 0.000, C 0.000 }
gfCNCPoint3[14420] = {X 421.1882, Y 17.5010, Z -4.6667, A 0.000, B 0.000, C 0.000 }
gfCNCPoint3[14421] = {X 420.5403, Y 18.3844, Z -4.6667, A 0.000, B 0.000, C 0.000 }
gfCNCPoint3[14422] = {X 419.9512, Y 19.3081, Z -4.6667, A 0.000, B 0.000, C 0.000 }
gfCNCPoint3[14423] = {X 412.1070, Y 31.9252, Z -4.6667, A 0.000, B 0.000, C 0.000 }
gfCNCPoint3[14424] = {X 412.1076, Y 40.6518, Z -4.6667, A 0.000, B 0.000, C 0.000 }
gfCNCPoint3[14425] = {X 412.7493, Y 41.4084, Z -4.6667, A 0.000, B 0.000, C 0.000 }
gfCNCPoint3[14426] = {X 413.2291, Y 42.2767, Z -4.6667, A 0.000, B 0.000, C 0.000 }
gfCNCPoint3[14427] = {X 413.5282, Y 43.2226, Z -4.6667, A 0.000, B 0.000, C 0.000 }
gfCNCPoint3[14428] = {X 413.6347, Y 44.2089, Z -4.6667, A 0.000, B 0.000, C 0.000 }
gfCNCPoint3[14429] = {X 413.6347, Y 45.0000, Z -4.6667, A 0.000, B 0.000, C 0.000 }
gfCNCPoint3[14430] = {X 413.6249, Y 45.3090, Z -4.6667, A 0.000, B 0.000, C 0.000 }
gfCNCPoint3[14431] = {X 413.5956, Y 45.6167, Z -4.6667, A 0.000, B 0.000, C 0.000 }
gfCNCPoint3[14432] = {X 413.3652, Y 46.5992, Z -4.6667, A 0.000, B 0.000, C 0.000 }
gfCNCPoint3[14433] = {X 412.9377, Y 47.5134, Z -4.6667, A 0.000, B 0.000, C 0.000 }
gfCNCPoint3[14434] = {X 412.3313, Y 48.3200, Z -4.6667, A 0.000, B 0.000, C 0.000 }
gfCNCPoint3[14435] = {X 411.9795, Y 47.9934, Z -4.6667, A 0.000, B 0.000, C 0.000 }
gfCNCPoint3[14436] = {X 411.3003, Y 48.5889, Z -4.6667, A 0.000, B 0.000, C 0.000 }
gfCNCPoint3[14437] = {X 410.5138, Y 49.0331, Z -4.6667, A 0.000, B 0.000, C 0.000 }
gfCNCPoint3[14438] = {X 409.6532, Y 49.3073, Z -4.6667, A 0.000, B 0.000, C 0.000 }
gfCNCPoint3[14439] = {X 408.7547, Y 49.4000, Z -4.6667, A 0.000, B 0.000, C 0.000 }
gfCNCPoint3[14440] = {X 402.3112, Y 49.4000, Z -4.6667, A 0.000, B 0.000, C 0.000 }
gfCNCPoint3[14441] = {X 401.3321, Y 49.2897, Z -4.6667, A 0.000, B 0.000, C 0.000 }
gfCNCPoint3[14442] = {X 400.4021, Y 48.9643, Z -4.6667, A 0.000, B 0.000, C 0.000 }
gfCNCPoint3[14443] = {X 399.5678, Y 48.4400, Z -4.6667, A 0.000, B 0.000, C 0.000 }
gfCNCPoint3[14444] = {X 398.8711, Y 47.7433, Z -4.6667, A 0.000, B 0.000, C 0.000 }
gfCNCPoint3[14445] = {X 398.3469, Y 46.9091, Z -4.6667, A 0.000, B 0.000, C 0.000 }
gfCNCPoint3[14446] = {X 398.0215, Y 45.9791, Z -4.6667, A 0.000, B 0.000, C 0.000 }
gfCNCPoint3[14447] = {X 397.9112, Y 45.0000, Z -4.6667, A 0.000, B 0.000, C 0.000 }
gfCNCPoint3[14448] = {X 397.9116, Y 44.1518, Z -4.6667, A 0.000, B 0.000, C 0.000 }
gfCNCPoint3[14449] = {X 398.0215, Y 43.2300, Z -4.6667, A 0.000, B 0.000, C 0.000 }
gfCNCPoint3[14450] = {X 398.3223, Y 42.3519, Z -4.6667, A 0.000, B 0.000, C 0.000 }
